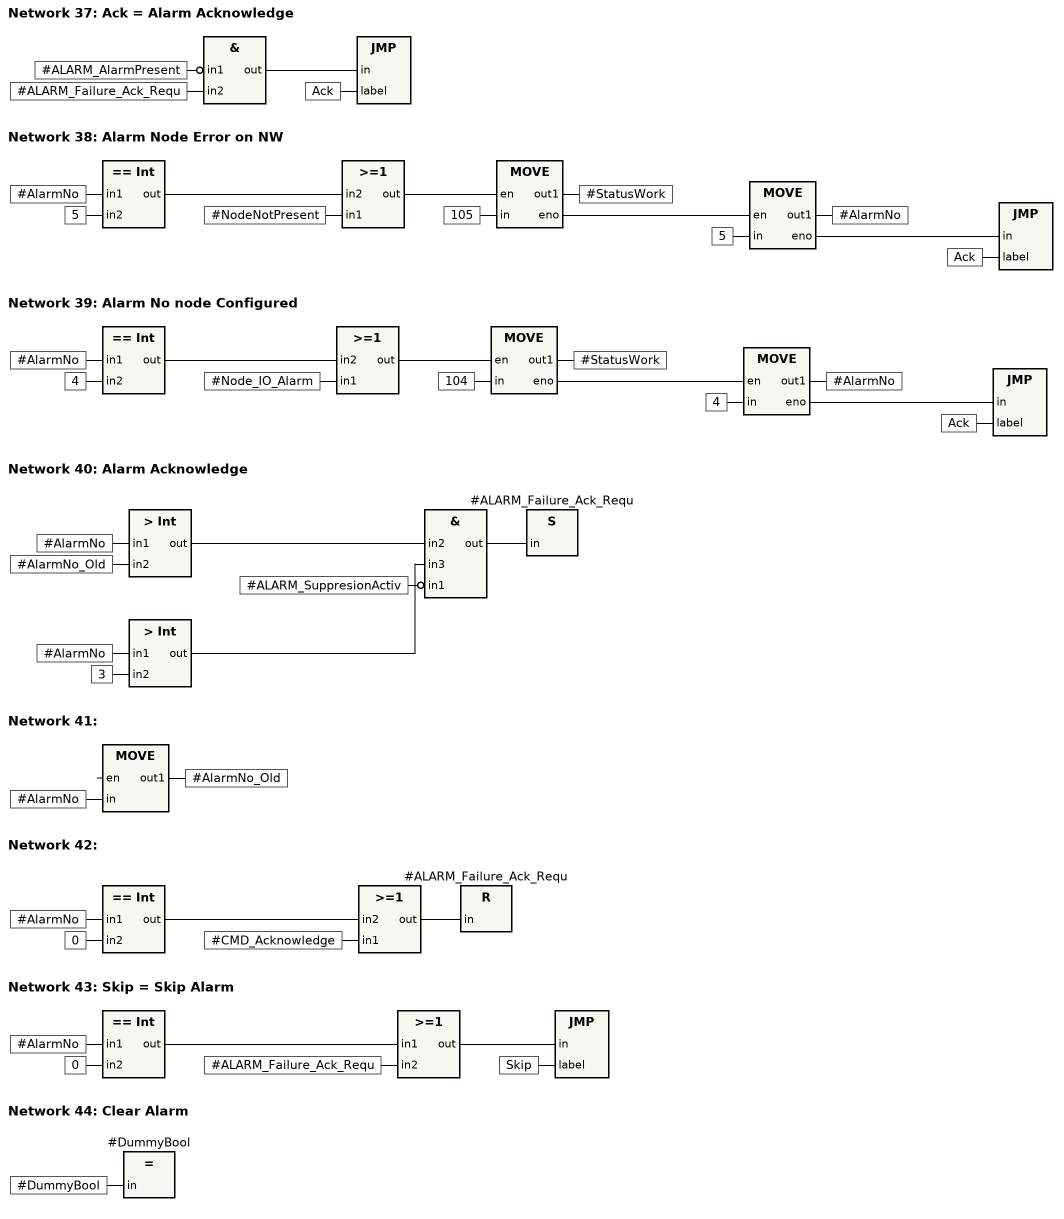
   IF NOT #ALARM_AlarmPresent AND #ALARM_Failure_Ack_Requ THEN GOTO Ack; END_IF;
END_REGION

REGION Network 38: Alarm Node Error on NW
   // ENO of a box is taken as its EN; it also drops when the box reports an error
   #_w1 := (#AlarmNo = 5) OR #NodeNotPresent;
   IF #_w1 THEN
       #StatusWork := 105;
       #AlarmNo := 5;
       GOTO Ack;
   END_IF;
END_REGION

REGION Network 39: Alarm No node Configured
   // ENO of a box is taken as its EN; it also drops when the box reports an error
   #_w1 := (#AlarmNo = 4) OR #Node_IO_Alarm;
   IF #_w1 THEN
       #StatusWork := 104;
       #AlarmNo := 4;
       GOTO Ack;
   END_IF;
END_REGION

REGION Network 40: Alarm Acknowledge
   Ack:
   IF (#AlarmNo > #AlarmNo_Old) AND (#AlarmNo > 3) AND NOT #ALARM_SuppresionActiv THEN
       #ALARM_Failure_Ack_Requ := TRUE;
   END_IF;
END_REGION

REGION Network 41
   #AlarmNo_Old := #AlarmNo;
END_REGION

REGION Network 42
   IF (#AlarmNo = 0) OR #CMD_Acknowledge THEN #ALARM_Failure_Ack_Requ := FALSE; END_IF;
END_REGION

REGION Network 43: Skip = Skip Alarm
   IF (#AlarmNo = 0) OR #ALARM_Failure_Ack_Requ THEN GOTO Skip; END_IF;
END_REGION

REGION Network 44: Clear Alarm
   Clr:
   #DummyBool := #DummyBool;
END_REGION

REGION Network 45
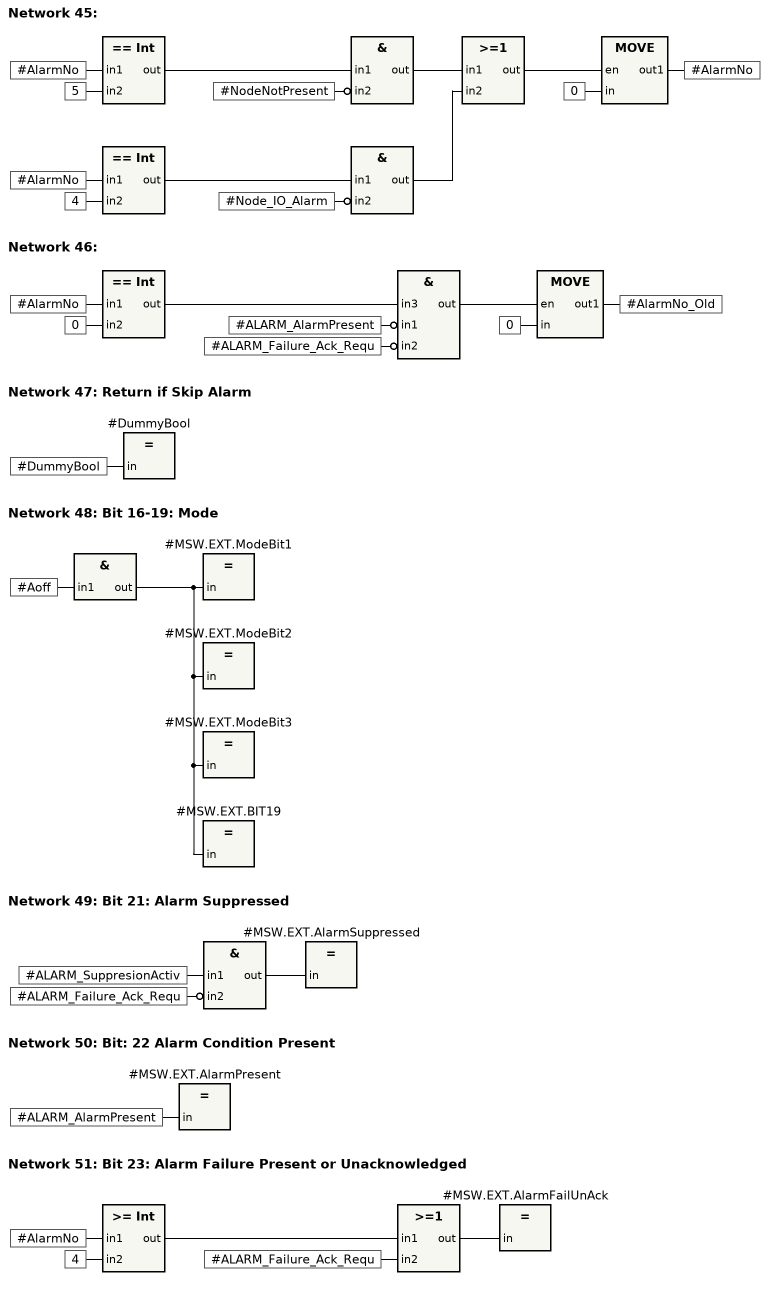
   IF ((#AlarmNo = 5) AND NOT #NodeNotPresent) OR ((#AlarmNo = 4) AND NOT #Node_IO_Alarm) THEN
       #AlarmNo := 0;
   END_IF;
END_REGION

REGION Network 46
   IF (#AlarmNo = 0) AND NOT #ALARM_AlarmPresent AND NOT #ALARM_Failure_Ack_Requ THEN
       #AlarmNo_Old := 0;
   END_IF;
END_REGION

REGION Network 47: Return if Skip Alarm
   Skip:
   #DummyBool := #DummyBool;
END_REGION

REGION Network 48: Bit 16-19: Mode
   // 0 = Auto
   // 1= Single Start
   // 2 = Manual
   // 3= Local
   // 4= Test Mode
   #MSW.EXT.ModeBit1 := #Aoff;
   #MSW.EXT.ModeBit2 := #Aoff;
   #MSW.EXT.ModeBit3 := #Aoff;
   #MSW.EXT.BIT19 := #Aoff;
END_REGION

REGION Network 49: Bit 21: Alarm Suppressed
   #MSW.EXT.AlarmSuppressed := #ALARM_SuppresionActiv AND NOT #ALARM_Failure_Ack_Requ;
END_REGION

REGION Network 50: Bit: 22 Alarm Condition Present
   #MSW.EXT.AlarmPresent := #ALARM_AlarmPresent;
END_REGION

REGION Network 51: Bit 23: Alarm Failure Present or Unacknowledged
   #MSW.EXT.AlarmFailUnAck := (#AlarmNo >= 4) OR #ALARM_Failure_Ack_Requ;
END_REGION

REGION Network 52: Bit 24: Alarm Warning Present Or Unacknowledged
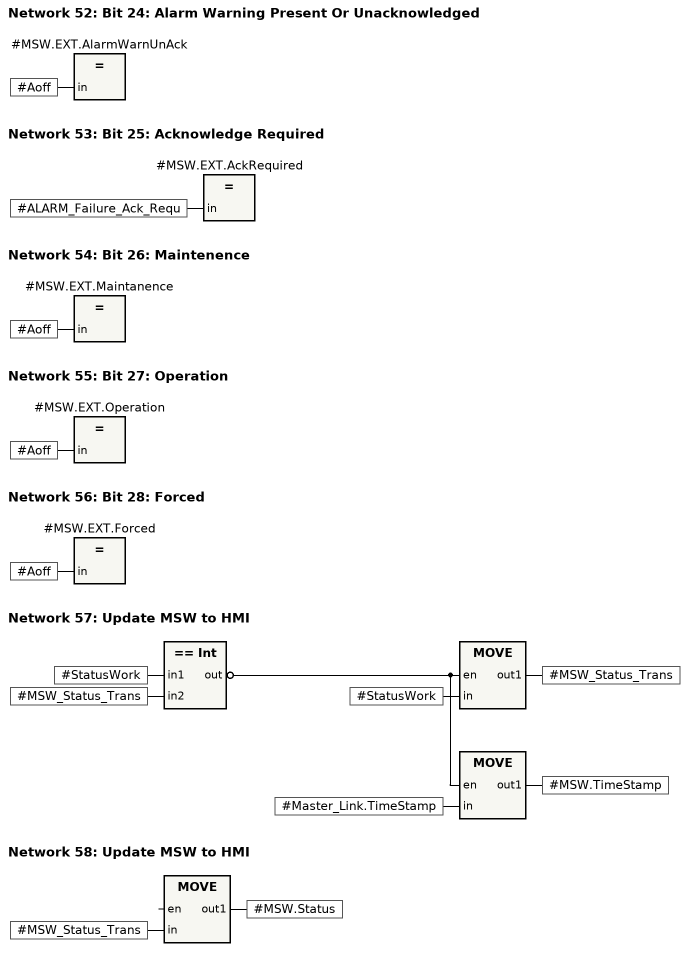
   #MSW.EXT.AlarmWarnUnAck := #Aoff;
END_REGION

REGION Network 53: Bit 25: Acknowledge Required
   #MSW.EXT.AckRequired := #ALARM_Failure_Ack_Requ;
END_REGION

REGION Network 54: Bit 26: Maintenence
   #MSW.EXT.Maintanence := #Aoff;
END_REGION

REGION Network 55: Bit 27: Operation
   #MSW.EXT.Operation := #Aoff;
END_REGION

REGION Network 56: Bit 28: Forced
   #MSW.EXT.Forced := #Aoff;
END_REGION

REGION Network 57: Update MSW to HMI
   #_w1 := NOT (#StatusWork = #MSW_Status_Trans);
   IF #_w1 THEN
       #MSW_Status_Trans := #StatusWork;
       #MSW.TimeStamp := #Master_Link.TimeStamp;
   END_IF;
END_REGION

REGION Network 58: Update MSW to HMI
   #MSW.Status := #MSW_Status_Trans;
END_REGION
END_FUNCTION_BLOCK

FUNCTION_BLOCK "ACESYS_SEND"   // FB225, FBD
TITLE = ACESYS V8.0 - Build 003 - SEND FUNCTION BLOCK
{ S7_Optimized_Access := 'TRUE' }
VERSION : 0.1
   VAR_INPUT
      Primary_EN : Bool;   // Enable Primary Link
      Primary_ID : Word;   // Valid from W#16#0001 to W#16#0FFF
      Primary_DEV_ID : Byte;   // 1 = Onboard (X1), 2 = Onboard (X2), 3 = Onboard (X3), 10 = External Cards
      Primary_ACT : Bool;   // ACTIVE=1; PASSIVE=0
      Primary_IP_ADDR1 : Int;   // Primary IP Address
      Primary_IP_ADDR2 : Int;   // Primary IP Address
      Primary_IP_ADDR3 : Int;   // Primary IP Address
      Primary_IP_ADDR4 : Int;   // Primary IP Address
      Primary_LOC_RS : Byte := BYTE#16#02;   // Primary Local Rack/Slot
      Primary_CP_RS : Byte;   // Primary CP Rack/Slot
      Primary_REM_RS : Byte := BYTE#16#02;   // Primary Remote Rack/Slot
      Secondary_EN : Bool;   // Enable Secondary Link
      Secondary_ID : Word;   // Valid from W#16#0001 to W#16#0FFF
      Secondary_DEV_ID : Byte;   // B#16#01-IM151-8PN, #02-CPU31x-2PN/DP, #03-CPU319-3PN/DP, #05-CPU41x-3PN/DP
      Secondary_ACT : Bool;
      Secondary_IP_ADDR1 : Int;   // Secondary IP Address
      Secondary_IP_ADDR2 : Int;   // Secondary IP Address
      Secondary_IP_ADDR3 : Int;   // Secondary IP Address
      Secondary_IP_ADDR4 : Int;   // Secondary IP Address
      Secondary_LOC_RS : Byte := BYTE#16#02;   // Secondary Local Rack/Slot
      Secondary_CP_RS : Byte;   // Secondary CP Rack/Slot
      Secondary_REM_RS : Byte := BYTE#16#02;   // Secondary Remote Rack/Slot
      DATA : "ACESYS_PlcToPLC";
      MASTER_LINK : "ACESYS_MASTER_LINK";
   END_VAR
   VAR_OUTPUT
      Primary_Comm_OK : Bool;   // Primary Communication OK
      Primary_Conn_St : Word;   // Primary Connection Status
      Primary_Send_St : Word;   // Primary Send Status
      Secondary_Comm_Ok : Bool;   // Secondary Communication OK
      Secondary_Conn_St : Word;   // Secondary Connection Status
      Secondary_Send_St : Word;   // Secondary Send Status
      MSW : "ACESYS_HMI_STAT_32T";
   END_VAR
   VAR
      BlockInfo : Struct
         Ace_Version : Int;   // Acesys Block Version Number
         Ace_BuildNo : Int;   // Acesys Block Build Number
         DB_Number : Int;   // Block Instance DB Number
      END_STRUCT;
      FP_CMD : Struct   // Faceplate Commands
         Spare_08 : Bool;
         Spare_09 : Bool;
         Spare_10 : Bool;
         Spare_11 : Bool;
         Spare_12 : Bool;
         Spare_13 : Bool;
         Spare_14 : Bool;
         AckAlarm : Bool;   // Alarm Acknowledge
         Spare_00 : Bool;
         Spare_01 : Bool;
         Spare_02 : Bool;
         Spare_03 : Bool;
         Spare_04 : Bool;
         Spare_05 : Bool;
         Spare_06 : Bool;
         Spare_07 : Bool;
      END_STRUCT;
      PRIM_T_SEND : TSEND;
      PRIM_T_CONN : TCON;
      PRIM_T_DISC : TDISCON;
      PRIM_T_PARAM : TCON_IP_RFC;
      PRIM_CONN_DATA : Struct
         REGISTERED : Bool;
         CONN_DONE : Bool;
         CONN_BUSY : Bool;
         CONN_ERROR : Bool;
         CONN_SETA : Bool;
         DISCONNECT : Bool;
         CONN_STATUS : Word;
         STATUS_SAV : Int;
         SEND_REQ : Bool;
         SEND_DONE : Bool;
         SEND_BUSY : Bool;
         SEND_ERROR : Bool;
         SEND_REQ_P : Bool;
         SEND_REQ_I : Bool;
         SEND_STATUS : Word;
         ABORT_REQ : Bool;
         ABORT_DONE : Bool;
         ABORT_BUSY : Bool;
         ABORT_ERROR : Bool;
         ABORT_REQ_I : Bool;
         ABORT_REQ_P : Bool;
         ABORT_STATUS : Word;
      END_STRUCT;
      SEC_T_SEND : TSEND;
      SEC_T_CONN : TCON;
      SEC_T_DISC : TDISCON;
      SEC_T_PARAM : TCON_IP_RFC;
      SEC_CONN_DATA : Struct
         REGISTERED : Bool;
         CONN_DONE : Bool;
         CONN_BUSY : Bool;
         CONN_ERROR : Bool;
         CONN_SETA : Bool;
         DISCONNECT : Bool;
         CONN_STATUS : Word;
         STATUS_SAV : Int;
         SEND_REQ : Bool;
         SEND_DONE : Bool;
         SEND_BUSY : Bool;
         SEND_ERROR : Bool;
         SEND_REQ_P : Bool;
         SEND_REQ_I : Bool;
         SEND_STATUS : Word;
         ABORT_REQ : Bool;
         ABORT_DONE : Bool;
         ABORT_BUSY : Bool;
         ABORT_ERROR : Bool;
         ABORT_REQ_I : Bool;
         ABORT_REQ_P : Bool;
         ABORT_STATUS : Word;
      END_STRUCT;
      TSAP16 : String[16];
      ID AT TSAP16 : Array[1..18] of Byte;
      Prim_String : String[16];
      Sec_String : String[16];
      Prim_INIT_COM : Bool;
      Sec_INIT_COM : Bool;
      Prim_En_ONS : Bool;
      Sec_En_ONS : Bool;
      Prim_Enabled_ONS : Bool;
      Sec_Enabled_ONS : Bool;
      SPECIFIED : Bool;
      Prim_ReCon_Active : Bool;   // Reconection Acive
      Sec_ReCon_Active : Bool;   // Reconection Acive
      Prim_SendReq_Dn : Bool;
      Sec_SendReq_Dn : Bool;
      Prim_EN : Bool;
      Sec_EN : Bool;
      Spare01 : Bool;
      Spare02 : Bool;
      Spare03 : Bool;
      Primary_ID_Old : Word;
      Secondary_ID_Old : Word;
      Prim_Con_TMR : TON_TIME;
      Prim_Del_ReCon : TON_TIME;   // Delay Before Auto ReConect
      Sec_Con_TMR : TON_TIME;
      Sec_Del_ReCon : TON_TIME;   // Delay Before Auto ReConect
      Prim_Com_OK : TON_TIME;
      Sec_Com_OK : TON_TIME;
      Prim_SendDelay : TON_TIME;
      Sec_SendDelay : TON_TIME;
      PRIM_EXT_HWID : GEOADDR;
      SEC_EXT_HWID : GEOADDR;
   END_VAR
   VAR_TEMP
      Aon : Bool;
      LOC_LEN : Int;
      REM_LEN : Int;
      TMP_INT : Int;
      LOC_RS : Int;
      TMP_RS : Int;
      TMP_DEV : Int;
      DummyBool : Bool;
      DummyDWord : DWord;
      DummyDInt : DInt;
      RET : Int;
      UDT_Length : Int;
      t_Zero : Int;
      b_Zero : Array[0..1] of Byte;
      SEND_DATA_Tmp : "ACESYS_PlcToPLC";
   END_VAR
   VAR_TEMP   // added for the SCL form of the ladder/FBD networks
      _w1 : Bool;
      _w2 : Bool;
      _w3 : Bool;
   END_VAR
BEGIN

REGION Network 1: Acesys Send Function Block based on Open Communication standard
   // Acesys Send Function Block based on Open Communication standard blocks FB63 and 
   // FB65 for ISO-on-TCP
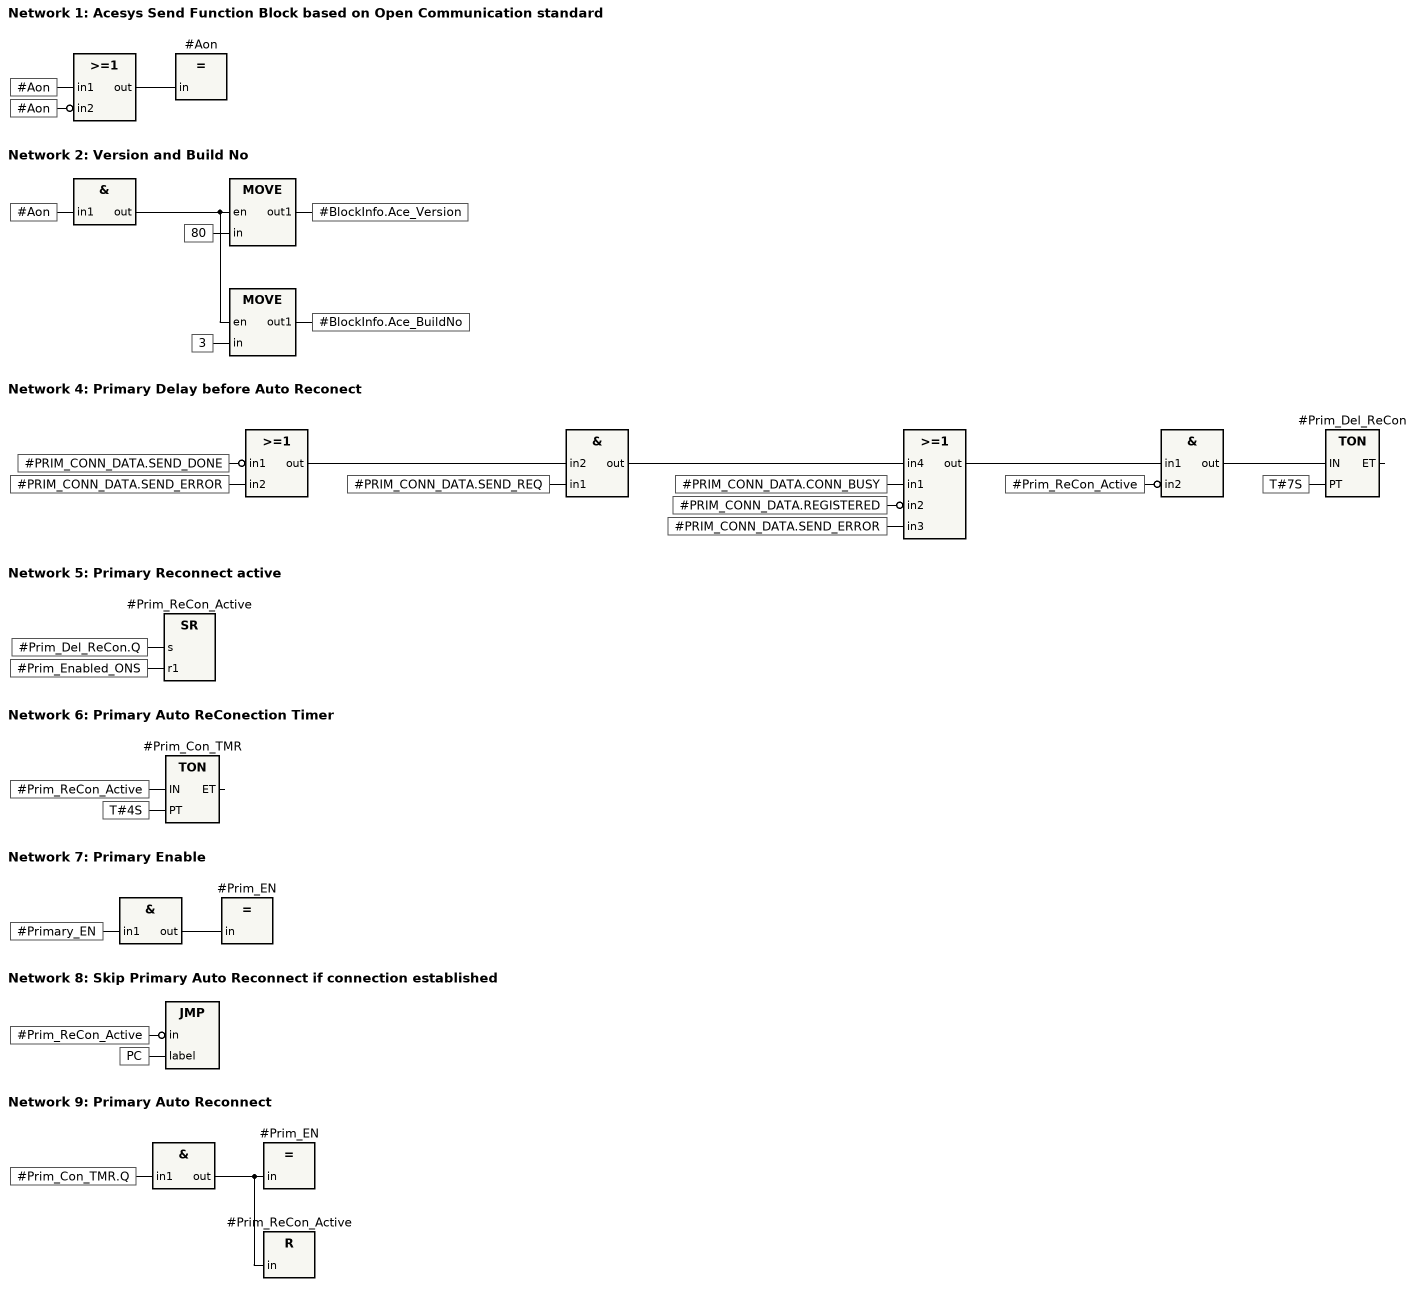
   #Aon := #Aon OR NOT #Aon;
END_REGION

REGION Network 2: Version and Build No
   IF #Aon THEN
       #BlockInfo.Ace_Version := 80;
       #BlockInfo.Ace_BuildNo := 3;
   END_IF;
END_REGION

REGION Network 3 (STL): Instance DB Number to Faceplate
         L     DINO;
         T     #BlockInfo.DB_Number;
END_REGION

REGION Network 4: Primary Delay before Auto Reconect
   #Prim_Del_ReCon(IN := (((NOT #PRIM_CONN_DATA.SEND_DONE OR #PRIM_CONN_DATA.SEND_ERROR) AND #PRIM_CONN_DATA.SEND_REQ) OR #PRIM_CONN_DATA.CONN_BUSY OR NOT #PRIM_CONN_DATA.REGISTERED OR #PRIM_CONN_DATA.SEND_ERROR) AND NOT #Prim_ReCon_Active,   // TON
                   PT := T#7S);
END_REGION

REGION Network 5: Primary Reconnect active
   IF #Prim_Del_ReCon.Q THEN
       #Prim_ReCon_Active := TRUE;   // SR flip-flop
   END_IF;
   IF #Prim_Enabled_ONS THEN #Prim_ReCon_Active := FALSE; END_IF;
END_REGION

REGION Network 6: Primary Auto ReConection Timer
   #Prim_Con_TMR(IN := #Prim_ReCon_Active, PT := T#4S);   // TON
END_REGION

REGION Network 7: Primary Enable
   #Prim_EN := #Primary_EN;
END_REGION

REGION Network 8: Skip Primary Auto Reconnect if connection established
   IF NOT #Prim_ReCon_Active THEN GOTO PC; END_IF;
END_REGION

REGION Network 9: Primary Auto Reconnect
   #Prim_EN := #Prim_Con_TMR.Q;
   IF #Prim_Con_TMR.Q THEN #Prim_ReCon_Active := FALSE; END_IF;
END_REGION

REGION Network 10: Set initial connection bit - Primary Link
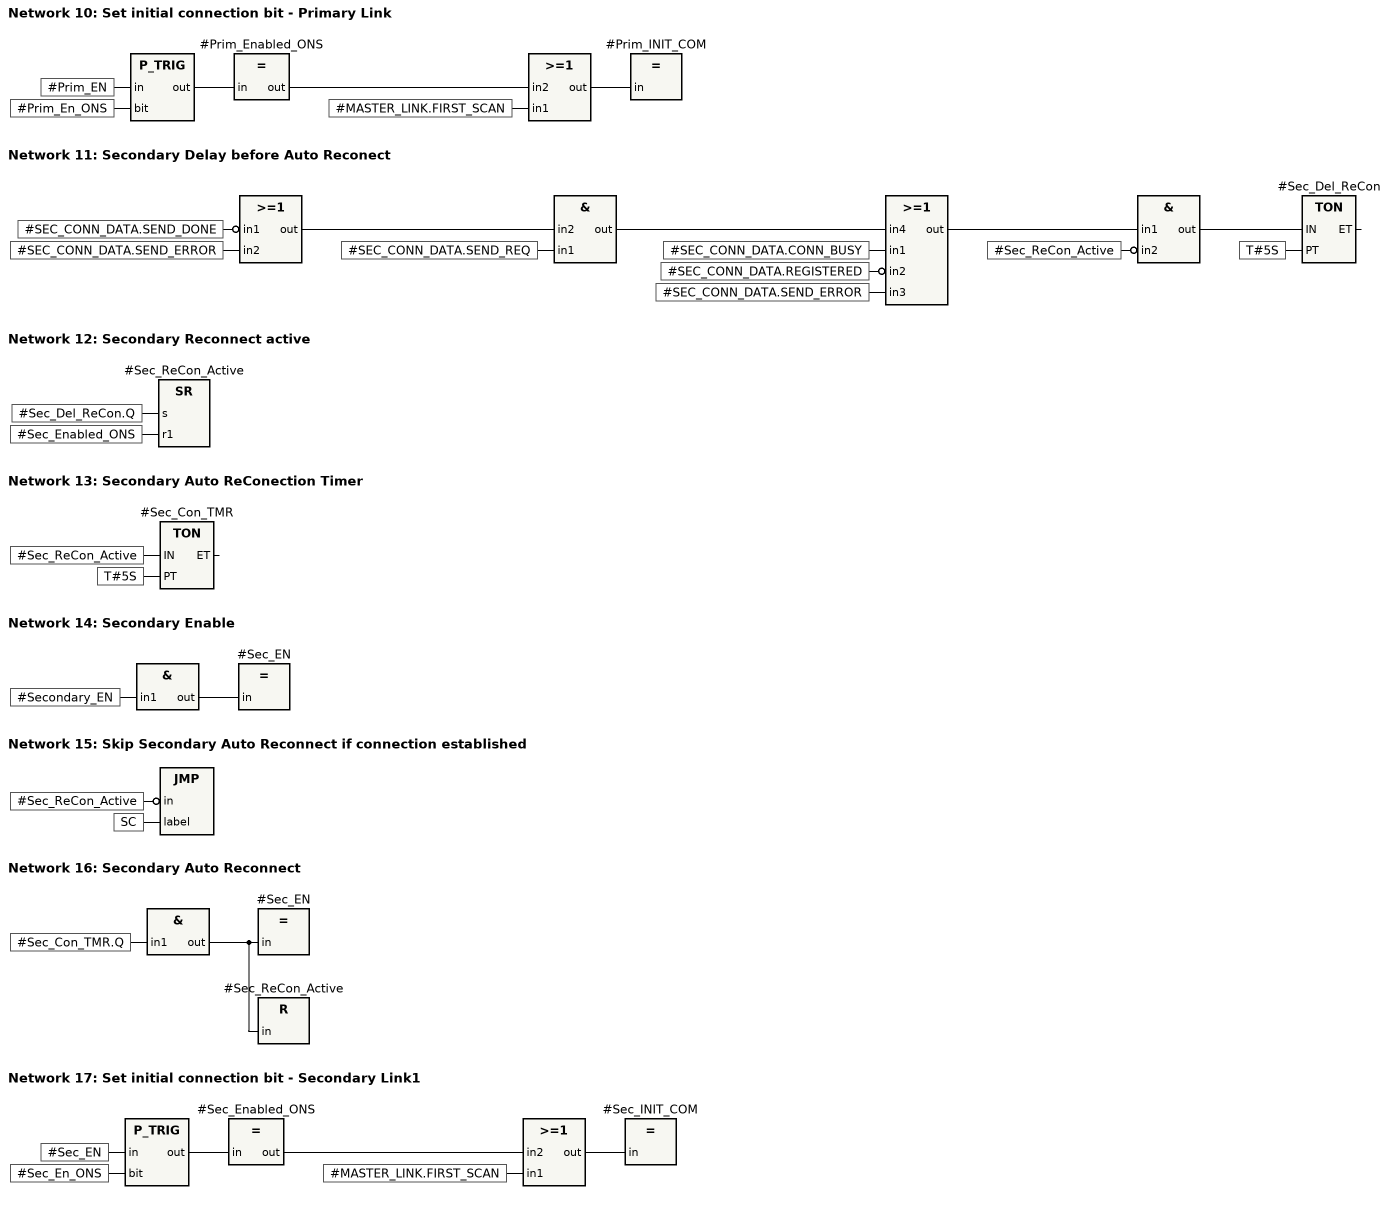
   PC:
   #_w1 := #Prim_EN AND NOT #Prim_En_ONS;   // rising edge
   #Prim_En_ONS := #Prim_EN;
   #Prim_Enabled_ONS := #_w1;
   #Prim_INIT_COM := #_w1 OR #MASTER_LINK.FIRST_SCAN;
END_REGION

REGION Network 11: Secondary Delay before Auto Reconect
   #Sec_Del_ReCon(IN := (((NOT #SEC_CONN_DATA.SEND_DONE OR #SEC_CONN_DATA.SEND_ERROR) AND #SEC_CONN_DATA.SEND_REQ) OR #SEC_CONN_DATA.CONN_BUSY OR NOT #SEC_CONN_DATA.REGISTERED OR #SEC_CONN_DATA.SEND_ERROR) AND NOT #Sec_ReCon_Active,   // TON
                  PT := T#5S);
END_REGION

REGION Network 12: Secondary Reconnect active
   IF #Sec_Del_ReCon.Q THEN
       #Sec_ReCon_Active := TRUE;   // SR flip-flop
   END_IF;
   IF #Sec_Enabled_ONS THEN #Sec_ReCon_Active := FALSE; END_IF;
END_REGION

REGION Network 13: Secondary Auto ReConection Timer
   #Sec_Con_TMR(IN := #Sec_ReCon_Active, PT := T#5S);   // TON
END_REGION

REGION Network 14: Secondary Enable
   #Sec_EN := #Secondary_EN;
END_REGION

REGION Network 15: Skip Secondary Auto Reconnect if connection established
   IF NOT #Sec_ReCon_Active THEN GOTO SC; END_IF;
END_REGION

REGION Network 16: Secondary Auto Reconnect
   #Sec_EN := #Sec_Con_TMR.Q;
   IF #Sec_Con_TMR.Q THEN #Sec_ReCon_Active := FALSE; END_IF;
END_REGION

REGION Network 17: Set initial connection bit - Secondary Link1
   SC:
   #_w1 := #Sec_EN AND NOT #Sec_En_ONS;   // rising edge
   #Sec_En_ONS := #Sec_EN;
   #Sec_Enabled_ONS := #_w1;
   #Sec_INIT_COM := #_w1 OR #MASTER_LINK.FIRST_SCAN;
END_REGION

REGION Network 18: Clear Bits to start initial connection and communication
   // Build002 - 27 March 2019 : Reset Condition PrimSendReq_Dn flag added
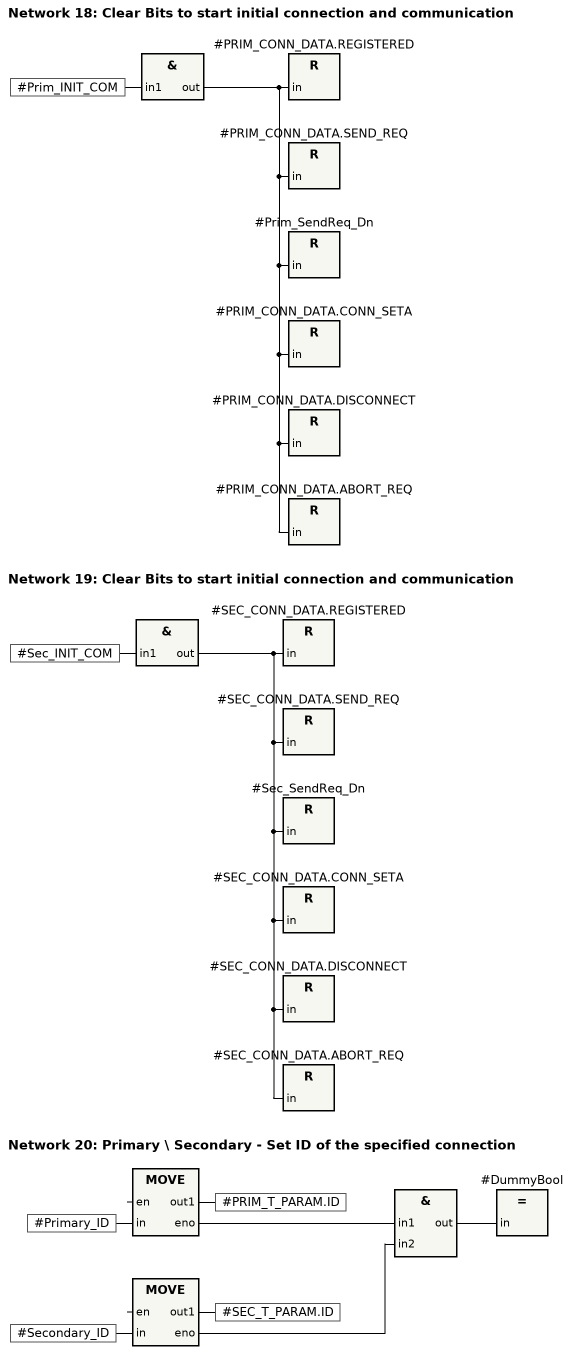
   IF #Prim_INIT_COM THEN
       #PRIM_CONN_DATA.REGISTERED := FALSE;
       #PRIM_CONN_DATA.SEND_REQ := FALSE;
       #Prim_SendReq_Dn := FALSE;
       #PRIM_CONN_DATA.CONN_SETA := FALSE;
       #PRIM_CONN_DATA.DISCONNECT := FALSE;
       #PRIM_CONN_DATA.ABORT_REQ := FALSE;
   END_IF;
END_REGION

REGION Network 19: Clear Bits to start initial connection and communication
   // Build002 - 27 March 2019 : Reset Condition SecSendReq_Dn flag added
   IF #Sec_INIT_COM THEN
       #SEC_CONN_DATA.REGISTERED := FALSE;
       #SEC_CONN_DATA.SEND_REQ := FALSE;
       #Sec_SendReq_Dn := FALSE;
       #SEC_CONN_DATA.CONN_SETA := FALSE;
       #SEC_CONN_DATA.DISCONNECT := FALSE;
       #SEC_CONN_DATA.ABORT_REQ := FALSE;
   END_IF;
END_REGION

REGION Network 20: Primary \ Secondary - Set ID of the specified connection
   // ENO of a box is taken as its EN; it also drops when the box reports an error
   #PRIM_T_PARAM.ID := #Primary_ID;
   #SEC_T_PARAM.ID := #Secondary_ID;
   #DummyBool := TRUE;
END_REGION

REGION Network 21: Primary \ Secondary - mode = 0x12 for ISO-on-TCP
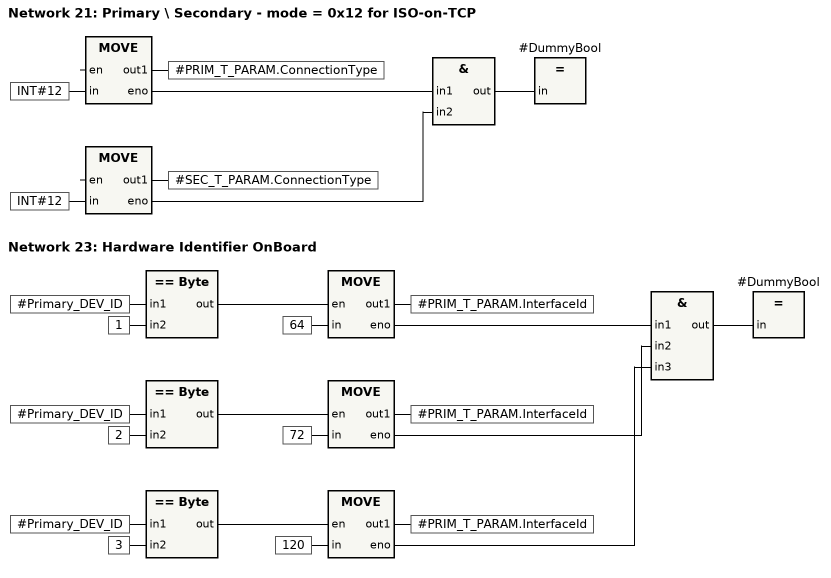
   // ENO of a box is taken as its EN; it also drops when the box reports an error
   #PRIM_T_PARAM.ConnectionType := INT#12;
   #SEC_T_PARAM.ConnectionType := INT#12;
   #DummyBool := TRUE;
END_REGION

REGION Network 22: <<<<<<<< PRIMARY >>>>>>>>
END_REGION

REGION Network 23: Hardware Identifier OnBoard
   // Build 003 viv-in 15 Feb 2022 -  X2 Port number corrected.
   #_w1 := #Primary_DEV_ID = 1;
   IF #_w1 THEN #PRIM_T_PARAM.InterfaceId := 64; END_IF;
   #_w2 := #Primary_DEV_ID = 2;
   IF #_w2 THEN #PRIM_T_PARAM.InterfaceId := 72; END_IF;
   #_w3 := #Primary_DEV_ID = 3;
   IF #_w3 THEN #PRIM_T_PARAM.InterfaceId := 120; END_IF;
   #DummyBool := #_w1 AND #_w2 AND #_w3;
END_REGION

REGION Network 24: Hardware Identifier External
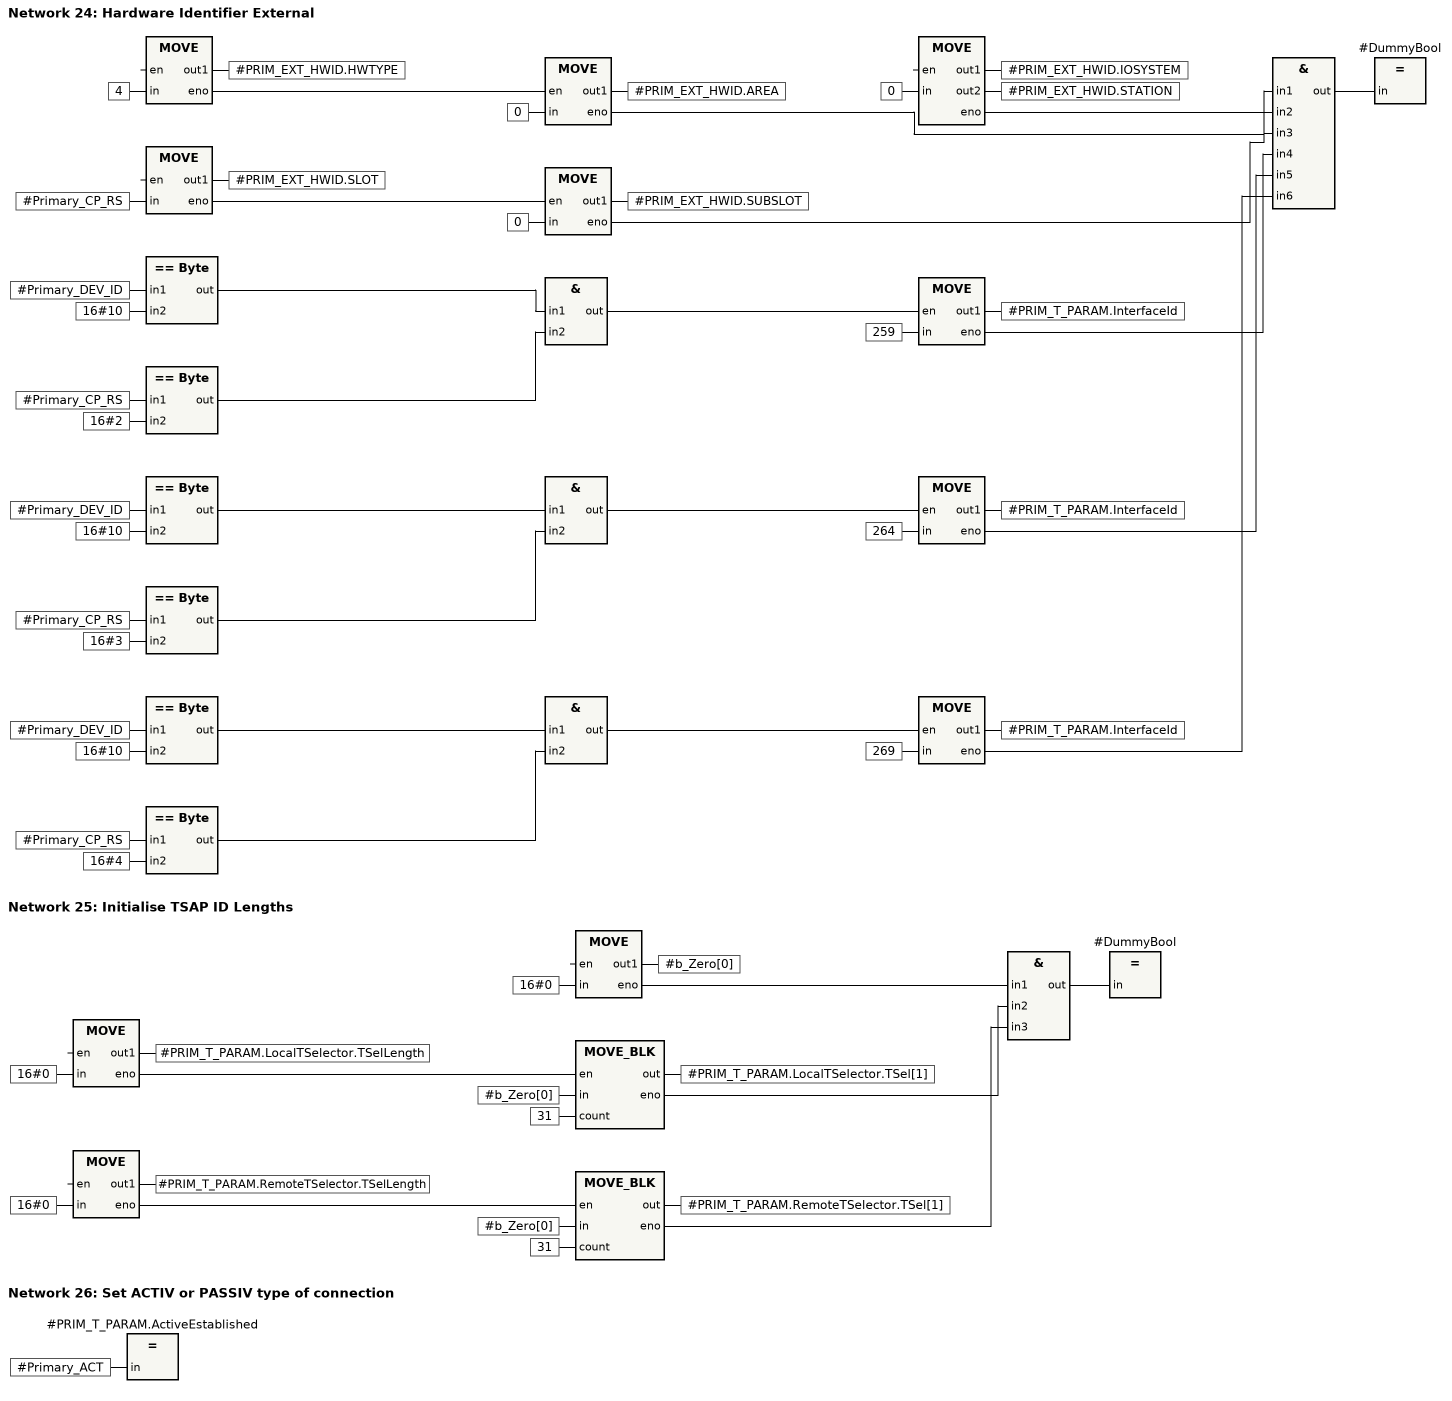
   #PRIM_EXT_HWID.HWTYPE := 4;
   #PRIM_EXT_HWID.AREA := 0;
   #PRIM_EXT_HWID.IOSYSTEM := 0;
   #PRIM_EXT_HWID.STATION := 0;
   #PRIM_EXT_HWID.SLOT := #Primary_CP_RS;
   #PRIM_EXT_HWID.SUBSLOT := 0;
   #_w1 := (#Primary_DEV_ID = 16#10) AND (#Primary_CP_RS = 16#2);
   IF #_w1 THEN #PRIM_T_PARAM.InterfaceId := 259; END_IF;
   #_w2 := (#Primary_DEV_ID = 16#10) AND (#Primary_CP_RS = 16#3);
   IF #_w2 THEN #PRIM_T_PARAM.InterfaceId := 264; END_IF;
   #_w3 := (#Primary_DEV_ID = 16#10) AND (#Primary_CP_RS = 16#4);
   IF #_w3 THEN #PRIM_T_PARAM.InterfaceId := 269; END_IF;
   #DummyBool := #_w1 AND #_w2 AND #_w3;
END_REGION

REGION Network 25: Initialise TSAP ID Lengths
   #b_Zero[0] := 16#0;
   #PRIM_T_PARAM.LocalTSelector.TSelLength := 16#0;
   MOVE_BLK(IN := #b_Zero[0], COUNT := 31, OUT => #PRIM_T_PARAM.LocalTSelector.TSel[1]);
   #PRIM_T_PARAM.RemoteTSelector.TSelLength := 16#0;
   MOVE_BLK(IN := #b_Zero[0], COUNT := 31, OUT => #PRIM_T_PARAM.RemoteTSelector.TSel[1]);
   #DummyBool := TRUE;
END_REGION

REGION Network 26: Set ACTIV or PASSIV type of connection
   // Receive Block Always Pasive
   #PRIM_T_PARAM.ActiveEstablished := #Primary_ACT;
END_REGION

REGION Network 27: Evaluate Rack/Slot being used for the leading bytes or none
   // 1) If R/S = 0 ---> no leading bytes are requested.
   // 2) If R/S # 0 ---> two leading bytes are required.
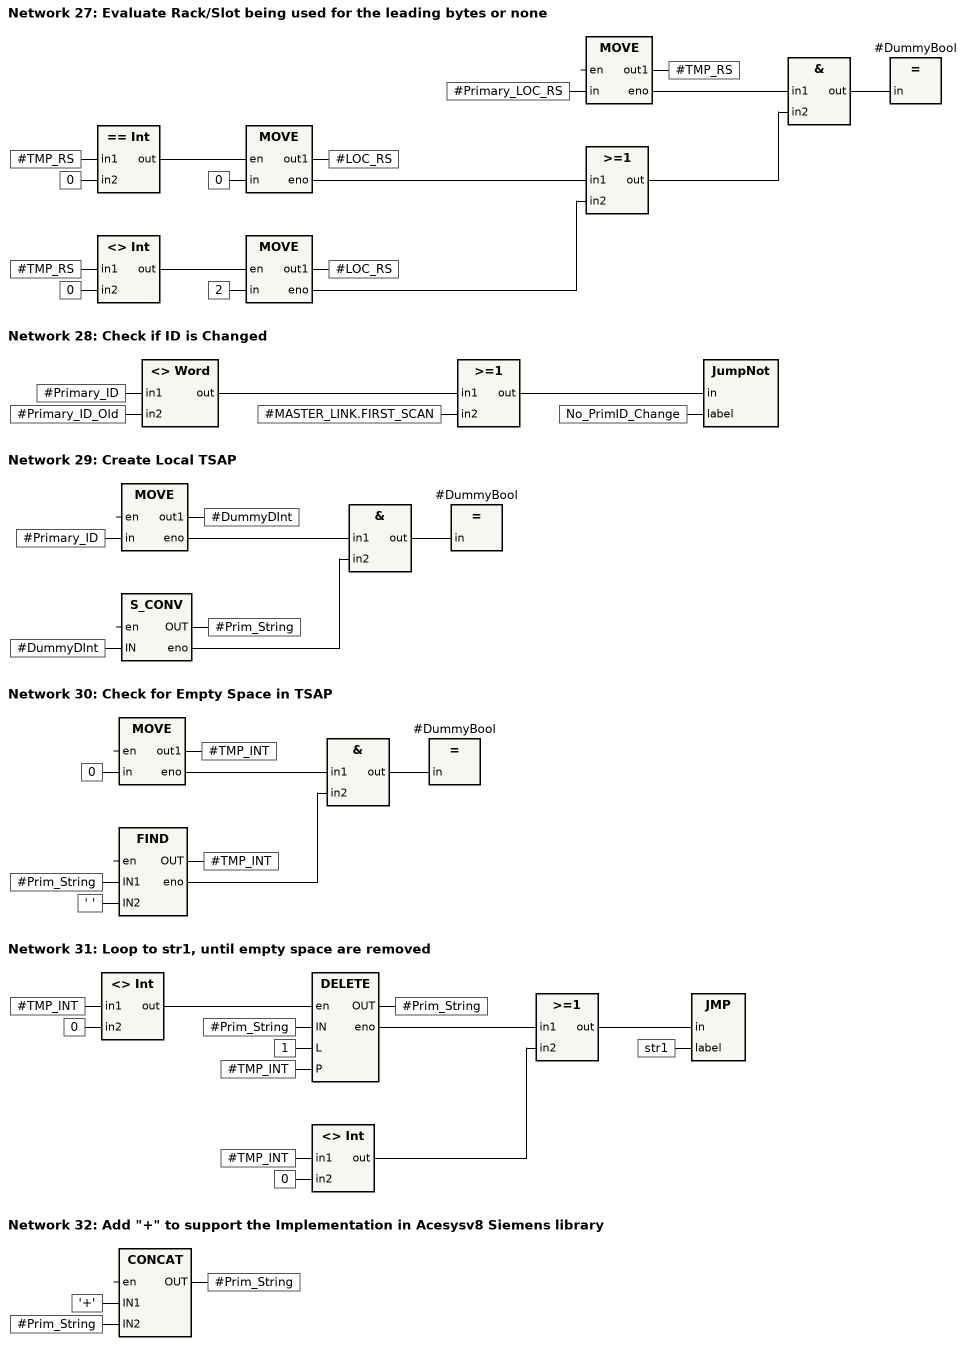
   // ENO of a box is taken as its EN; it also drops when the box reports an error
   #TMP_RS := #Primary_LOC_RS;
   #_w1 := #TMP_RS = 0;
   IF #_w1 THEN #LOC_RS := 0; END_IF;
   #_w2 := #TMP_RS <> 0;
   IF #_w2 THEN #LOC_RS := 2; END_IF;
   #DummyBool := #_w1 OR #_w2;
END_REGION

REGION Network 28: Check if ID is Changed
   // no SCL statement known for JumpNot: written as a call
   JumpNot(in := (#Primary_ID <> #Primary_ID_Old) OR #MASTER_LINK.FIRST_SCAN, label := No_PrimID_Change);
END_REGION

REGION Network 29: Create Local TSAP
   // Local TSAP = ID_Number
   // ENO of a box is taken as its EN; it also drops when the box reports an error
   #DummyDInt := #Primary_ID;
   #Prim_String := S_CONV(IN := #DummyDInt);
   #DummyBool := TRUE;
END_REGION

REGION Network 30: Check for Empty Space in TSAP
   str1:
   #TMP_INT := 0;
   #TMP_INT := FIND(IN1 := #Prim_String, IN2 := ' ');
   #DummyBool := TRUE;
END_REGION

REGION Network 31: Loop to str1, until empty space are removed
   #_w1 := #TMP_INT <> 0;
   IF #_w1 THEN #Prim_String := DELETE(IN := #Prim_String, L := 1, P := #TMP_INT); END_IF;
   IF #_w1 OR (#TMP_INT <> 0) THEN GOTO str1; END_IF;
END_REGION

REGION Network 32: Add "+" to support the Implementation in Acesysv8 Siemens library
   #Prim_String := CONCAT(IN1 := '+', IN2 := #Prim_String);
END_REGION

REGION Network 33: Set Primary_ID_Old Temp
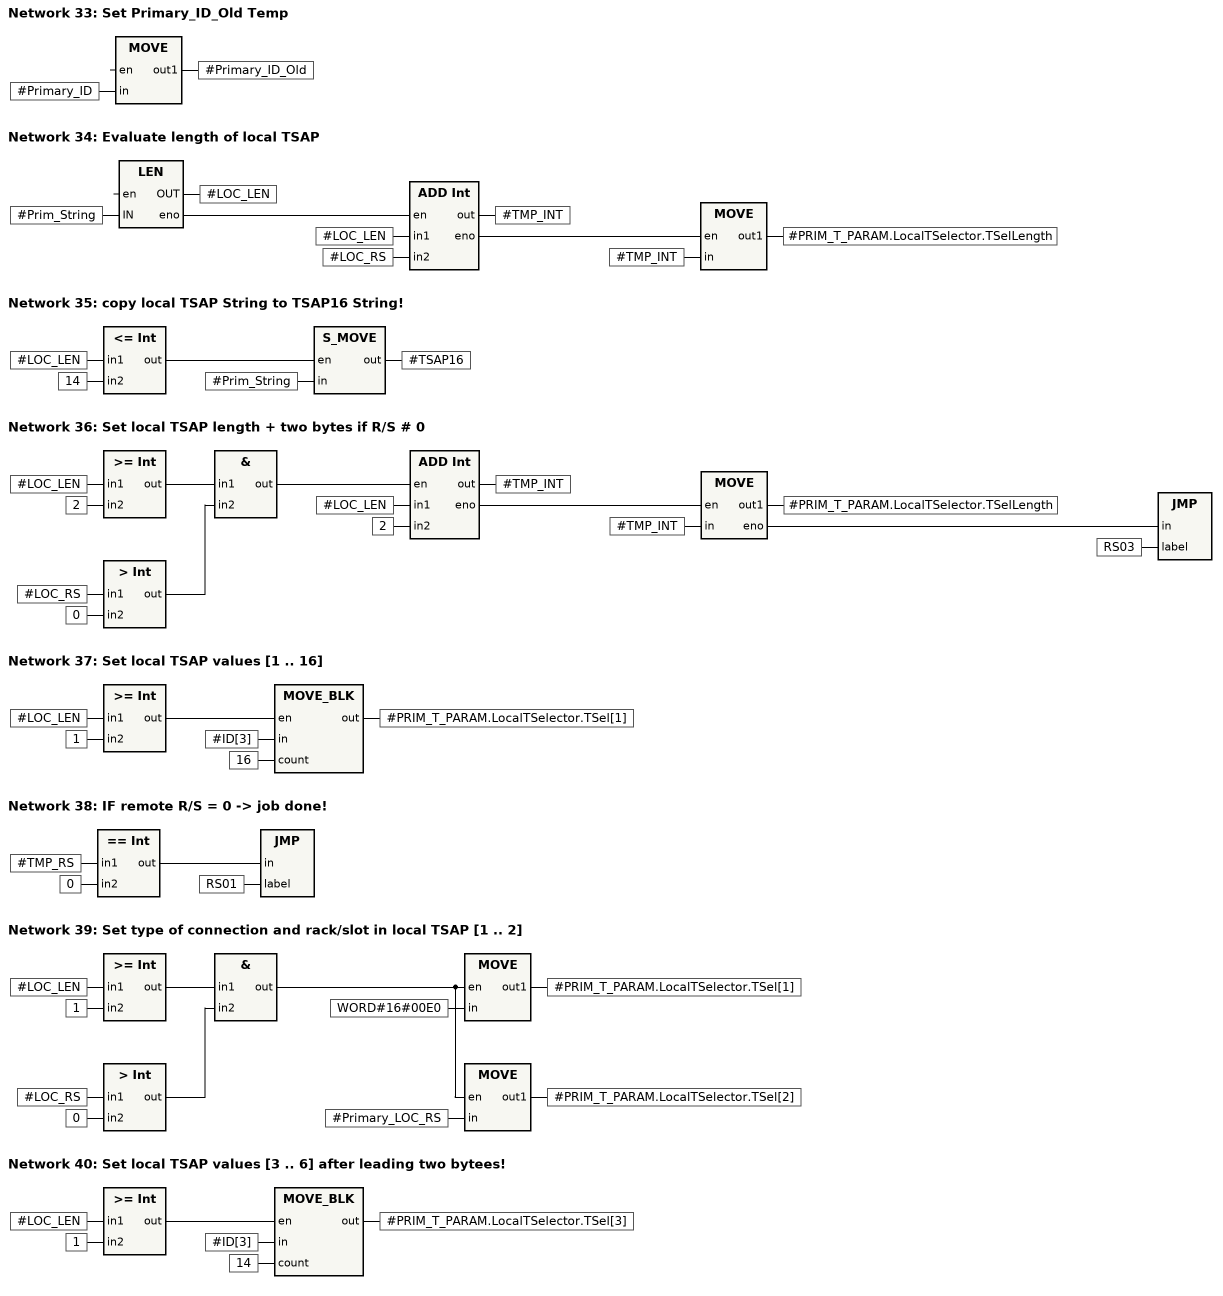
   No_PrimID_Change:
   #Primary_ID_Old := #Primary_ID;
END_REGION

REGION Network 34: Evaluate length of local TSAP
   // #TSAP.LOC_TSAP
   // ENO of a box is taken as its EN; it also drops when the box reports an error
   #LOC_LEN := LEN(IN := #Prim_String);
   #TMP_INT := #LOC_LEN + #LOC_RS;
   #PRIM_T_PARAM.LocalTSelector.TSelLength := #TMP_INT;
END_REGION

REGION Network 35: copy local TSAP String to TSAP16 String!
   // #TSAP.LOC_TSAP
   IF #LOC_LEN <= 14 THEN #TSAP16 := #Prim_String; END_IF;
END_REGION

REGION Network 36: Set local TSAP length + two bytes if R/S # 0
   // ENO of a box is taken as its EN; it also drops when the box reports an error
   #_w1 := (#LOC_LEN >= 2) AND (#LOC_RS > 0);
   IF #_w1 THEN
       #TMP_INT := #LOC_LEN + 2;
       #PRIM_T_PARAM.LocalTSelector.TSelLength := #TMP_INT;
       GOTO RS03;
   END_IF;
END_REGION

REGION Network 37: Set local TSAP values [1 .. 16]
   // Fill in the entire local TSAP (without leading bytes)
   IF #LOC_LEN >= 1 THEN
       MOVE_BLK(IN := #ID[3], COUNT := 16, OUT => #PRIM_T_PARAM.LocalTSelector.TSel[1]);
   END_IF;
END_REGION

REGION Network 38: IF remote R/S = 0 -> job done!
   IF #TMP_RS = 0 THEN GOTO RS01; END_IF;
END_REGION

REGION Network 39: Set type of connection and rack/slot in local TSAP [1 .. 2]
   // B#16#E0 -> type of connection 
   // B#16#02 -> rack/slot of CPU
   RS03:
   IF (#LOC_LEN >= 1) AND (#LOC_RS > 0) THEN
       #PRIM_T_PARAM.LocalTSelector.TSel[1] := WORD#16#00E0;
       #PRIM_T_PARAM.LocalTSelector.TSel[2] := #Primary_LOC_RS;
   END_IF;
END_REGION

REGION Network 40: Set local TSAP values [3 .. 6] after leading two bytees!
   IF #LOC_LEN >= 1 THEN
       MOVE_BLK(IN := #ID[3], COUNT := 14, OUT => #PRIM_T_PARAM.LocalTSelector.TSel[3]);
   END_IF;
END_REGION

REGION Network 41: REMOTE TSAP
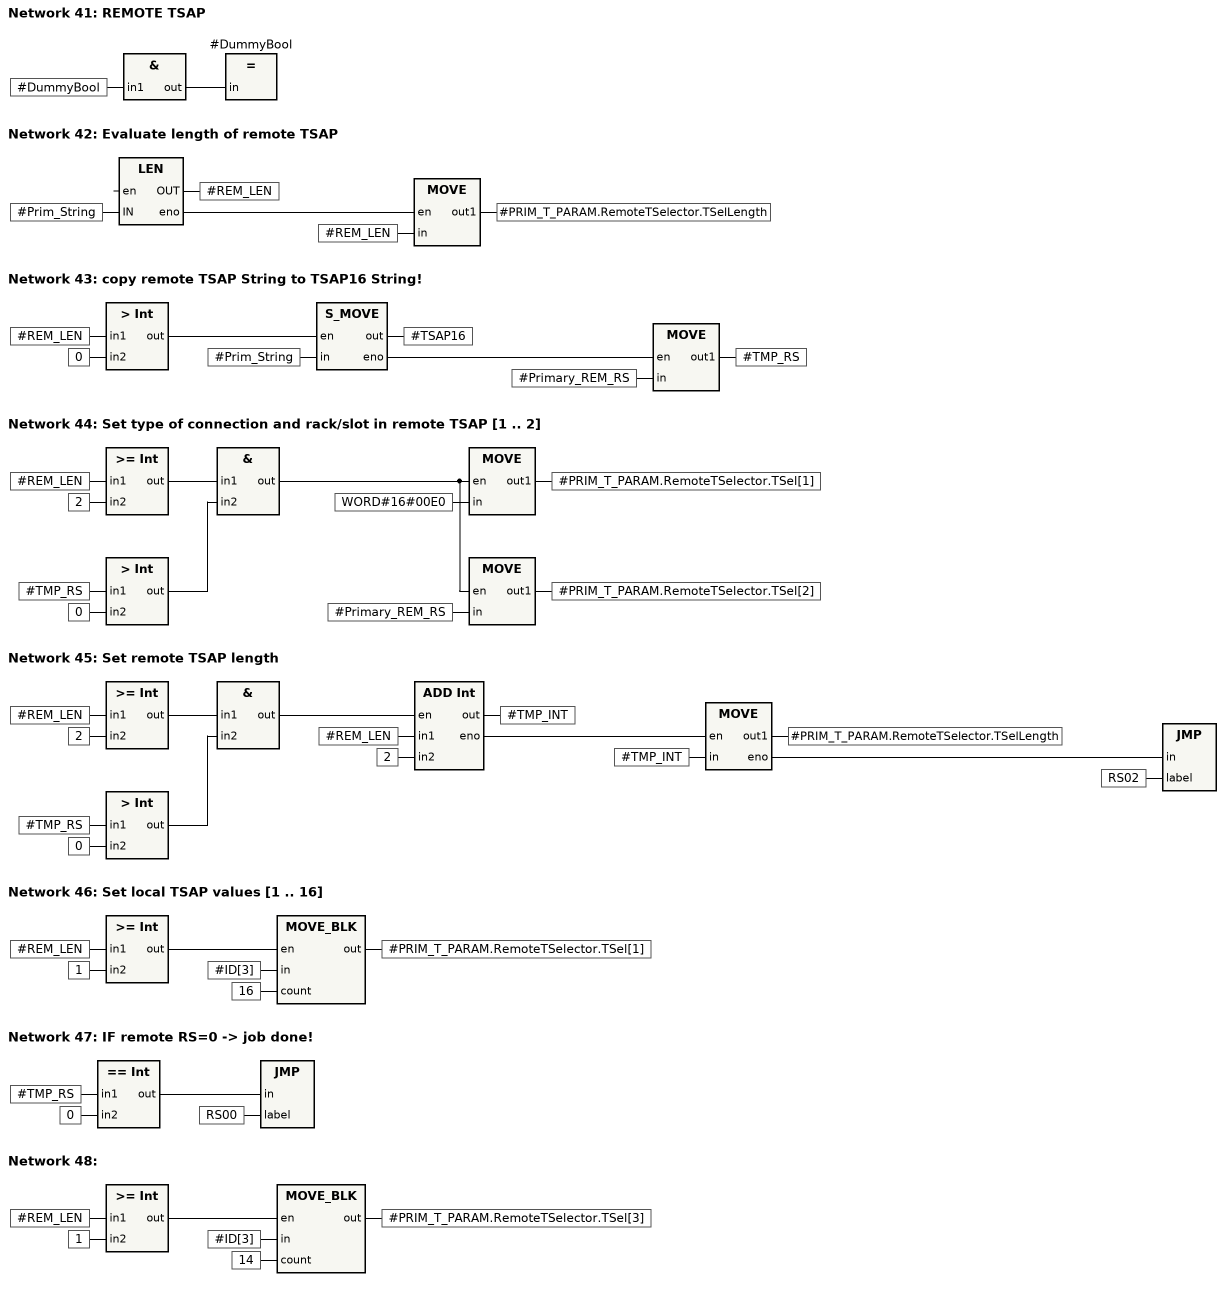
   RS01:
   #DummyBool := #DummyBool;
END_REGION

REGION Network 42: Evaluate length of remote TSAP
   // Remote TSAP = Local TSAP (DummyString1)
   #REM_LEN := LEN(IN := #Prim_String);
   #PRIM_T_PARAM.RemoteTSelector.TSelLength := #REM_LEN;
END_REGION

REGION Network 43: copy remote TSAP String to TSAP16 String!
   // Remote TSAP = Local TSAP (DummyString)
   IF #REM_LEN > 0 THEN
       #TSAP16 := #Prim_String;
       #TMP_RS := #Primary_REM_RS;
   END_IF;
END_REGION

REGION Network 44: Set type of connection and rack/slot in remote TSAP [1 .. 2]
   // B#16#E0 -> type of connection 
   // B#16#02 -> rack/slot of CPU
   IF (#REM_LEN >= 2) AND (#TMP_RS > 0) THEN
       #PRIM_T_PARAM.RemoteTSelector.TSel[1] := WORD#16#00E0;
       #PRIM_T_PARAM.RemoteTSelector.TSel[2] := #Primary_REM_RS;
   END_IF;
END_REGION

REGION Network 45: Set remote TSAP length
   // ENO of a box is taken as its EN; it also drops when the box reports an error
   #_w1 := (#REM_LEN >= 2) AND (#TMP_RS > 0);
   IF #_w1 THEN
       #TMP_INT := #REM_LEN + 2;
       #PRIM_T_PARAM.RemoteTSelector.TSelLength := #TMP_INT;
       GOTO RS02;
   END_IF;
END_REGION

REGION Network 46: Set local TSAP values [1 .. 16]
   // Fill in the entire local TSAP (without leading bytes)
   IF #REM_LEN >= 1 THEN
       MOVE_BLK(IN := #ID[3], COUNT := 16, OUT => #PRIM_T_PARAM.RemoteTSelector.TSel[1]);
   END_IF;
END_REGION

REGION Network 47: IF remote RS=0 -> job done!
   IF #TMP_RS = 0 THEN GOTO RS00; END_IF;
END_REGION

REGION Network 48
   RS02:
   IF #REM_LEN >= 1 THEN
       MOVE_BLK(IN := #ID[3], COUNT := 14, OUT => #PRIM_T_PARAM.RemoteTSelector.TSel[3]);
   END_IF;
END_REGION

REGION Network 49: Set length of the IP address if full-specified only !
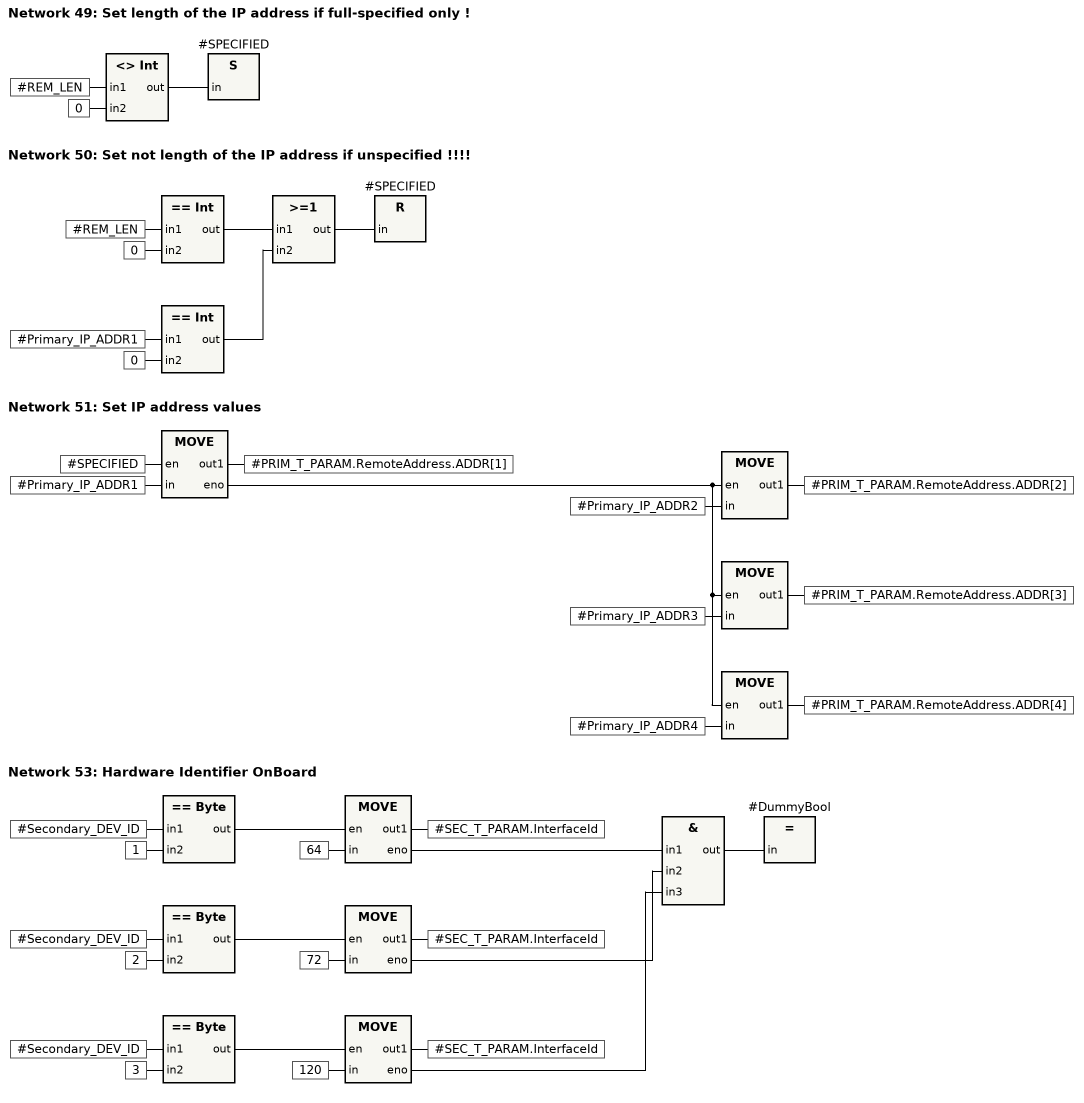
   RS00:
   IF #REM_LEN <> 0 THEN #SPECIFIED := TRUE; END_IF;
END_REGION

REGION Network 50: Set not length of the IP address if unspecified !!!!
   // The remote IP address must be zero if
   // 1) remote TSAP is unspecified, or
   // 2) IP address is set up with zero!
   IF (#REM_LEN = 0) OR (#Primary_IP_ADDR1 = 0) THEN #SPECIFIED := FALSE; END_IF;
END_REGION

REGION Network 51: Set IP address values
   // ENO of a box is taken as its EN; it also drops when the box reports an error
   IF #SPECIFIED THEN
       #PRIM_T_PARAM.RemoteAddress.ADDR[1] := #Primary_IP_ADDR1;
       #PRIM_T_PARAM.RemoteAddress.ADDR[2] := #Primary_IP_ADDR2;
       #PRIM_T_PARAM.RemoteAddress.ADDR[3] := #Primary_IP_ADDR3;
       #PRIM_T_PARAM.RemoteAddress.ADDR[4] := #Primary_IP_ADDR4;
   END_IF;
END_REGION

REGION Network 52: <<<<<<<<<<SECONDARY>>>>>>>>>>
END_REGION

REGION Network 53: Hardware Identifier OnBoard
   // Build 003 viv-in 15 Feb 2022 -  X2 Port number corrected.
   #_w1 := #Secondary_DEV_ID = 1;
   IF #_w1 THEN #SEC_T_PARAM.InterfaceId := 64; END_IF;
   #_w2 := #Secondary_DEV_ID = 2;
   IF #_w2 THEN #SEC_T_PARAM.InterfaceId := 72; END_IF;
   #_w3 := #Secondary_DEV_ID = 3;
   IF #_w3 THEN #SEC_T_PARAM.InterfaceId := 120; END_IF;
   #DummyBool := #_w1 AND #_w2 AND #_w3;
END_REGION

REGION Network 54: Hardware Identifier External
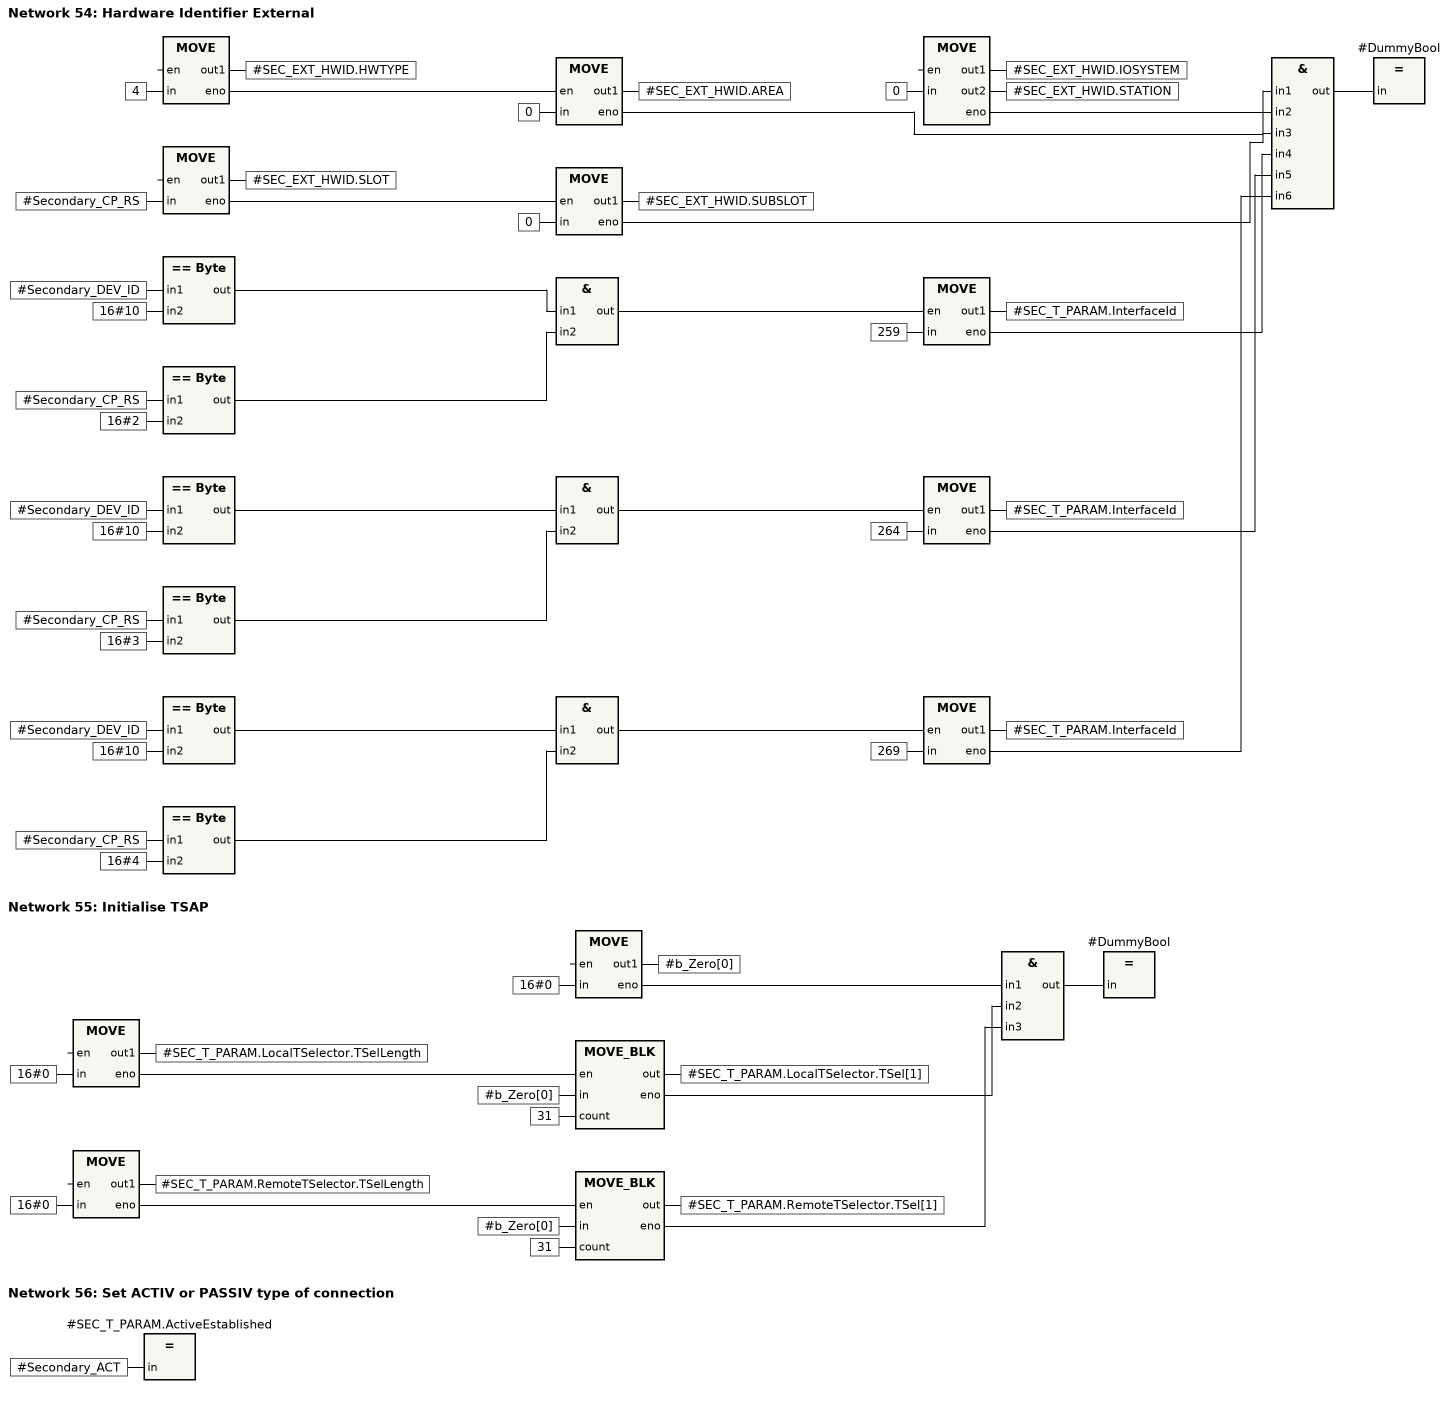
   #SEC_EXT_HWID.HWTYPE := 4;
   #SEC_EXT_HWID.AREA := 0;
   #SEC_EXT_HWID.IOSYSTEM := 0;
   #SEC_EXT_HWID.STATION := 0;
   #SEC_EXT_HWID.SLOT := #Secondary_CP_RS;
   #SEC_EXT_HWID.SUBSLOT := 0;
   #_w1 := (#Secondary_DEV_ID = 16#10) AND (#Secondary_CP_RS = 16#2);
   IF #_w1 THEN #SEC_T_PARAM.InterfaceId := 259; END_IF;
   #_w2 := (#Secondary_DEV_ID = 16#10) AND (#Secondary_CP_RS = 16#3);
   IF #_w2 THEN #SEC_T_PARAM.InterfaceId := 264; END_IF;
   #_w3 := (#Secondary_DEV_ID = 16#10) AND (#Secondary_CP_RS = 16#4);
   IF #_w3 THEN #SEC_T_PARAM.InterfaceId := 269; END_IF;
   #DummyBool := #_w1 AND #_w2 AND #_w3;
END_REGION

REGION Network 55: Initialise TSAP
   #b_Zero[0] := 16#0;
   #SEC_T_PARAM.LocalTSelector.TSelLength := 16#0;
   MOVE_BLK(IN := #b_Zero[0], COUNT := 31, OUT => #SEC_T_PARAM.LocalTSelector.TSel[1]);
   #SEC_T_PARAM.RemoteTSelector.TSelLength := 16#0;
   MOVE_BLK(IN := #b_Zero[0], COUNT := 31, OUT => #SEC_T_PARAM.RemoteTSelector.TSel[1]);
   #DummyBool := TRUE;
END_REGION

REGION Network 56: Set ACTIV or PASSIV type of connection
   // Send Block Always Active
   #SEC_T_PARAM.ActiveEstablished := #Secondary_ACT;
END_REGION

REGION Network 57: Evaluate Rack/Slot being used for the leading bytes or none
   // 1) If R/S = 0 ---> no leading bytes are requested.
   // 2) If R/S # 0 ---> two leading bytes are required.
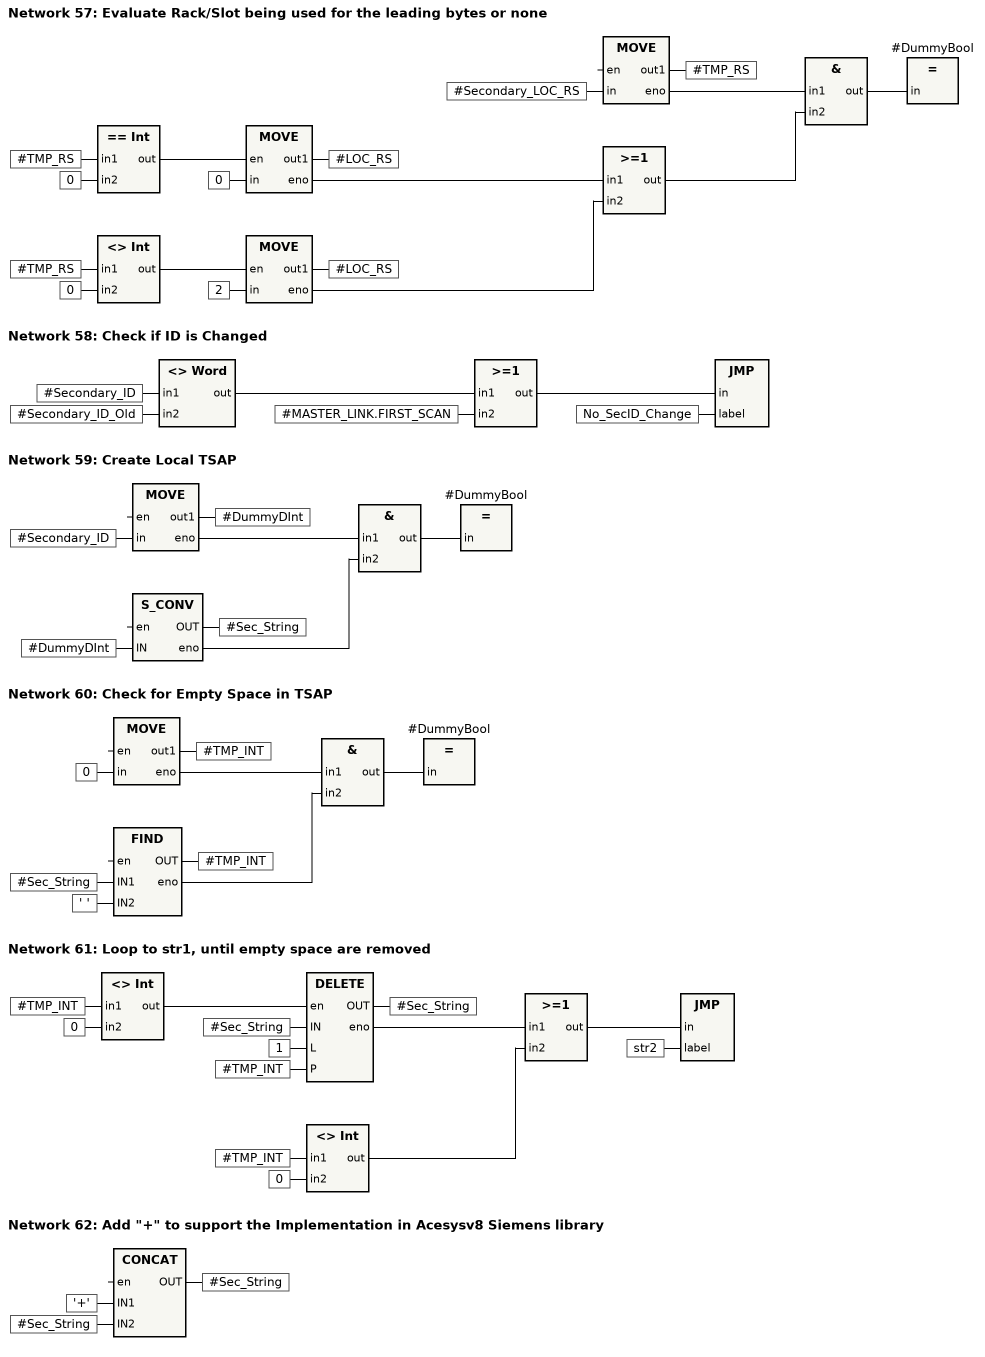
   // ENO of a box is taken as its EN; it also drops when the box reports an error
   #TMP_RS := #Secondary_LOC_RS;
   #_w1 := #TMP_RS = 0;
   IF #_w1 THEN #LOC_RS := 0; END_IF;
   #_w2 := #TMP_RS <> 0;
   IF #_w2 THEN #LOC_RS := 2; END_IF;
   #DummyBool := #_w1 OR #_w2;
END_REGION

REGION Network 58: Check if ID is Changed
   IF (#Secondary_ID <> #Secondary_ID_Old) OR #MASTER_LINK.FIRST_SCAN THEN GOTO No_SecID_Change; END_IF;
END_REGION

REGION Network 59: Create Local TSAP
   // Local TSAP = ID_Number
   // ENO of a box is taken as its EN; it also drops when the box reports an error
   #DummyDInt := #Secondary_ID;
   #Sec_String := S_CONV(IN := #DummyDInt);
   #DummyBool := TRUE;
END_REGION

REGION Network 60: Check for Empty Space in TSAP
   str2:
   #TMP_INT := 0;
   #TMP_INT := FIND(IN1 := #Sec_String, IN2 := ' ');
   #DummyBool := TRUE;
END_REGION

REGION Network 61: Loop to str1, until empty space are removed
   #_w1 := #TMP_INT <> 0;
   IF #_w1 THEN #Sec_String := DELETE(IN := #Sec_String, L := 1, P := #TMP_INT); END_IF;
   IF #_w1 OR (#TMP_INT <> 0) THEN GOTO str2; END_IF;
END_REGION

REGION Network 62: Add "+" to support the Implementation in Acesysv8 Siemens library
   #Sec_String := CONCAT(IN1 := '+', IN2 := #Sec_String);
END_REGION

REGION Network 63: Set Secondary_ID_Old Temp
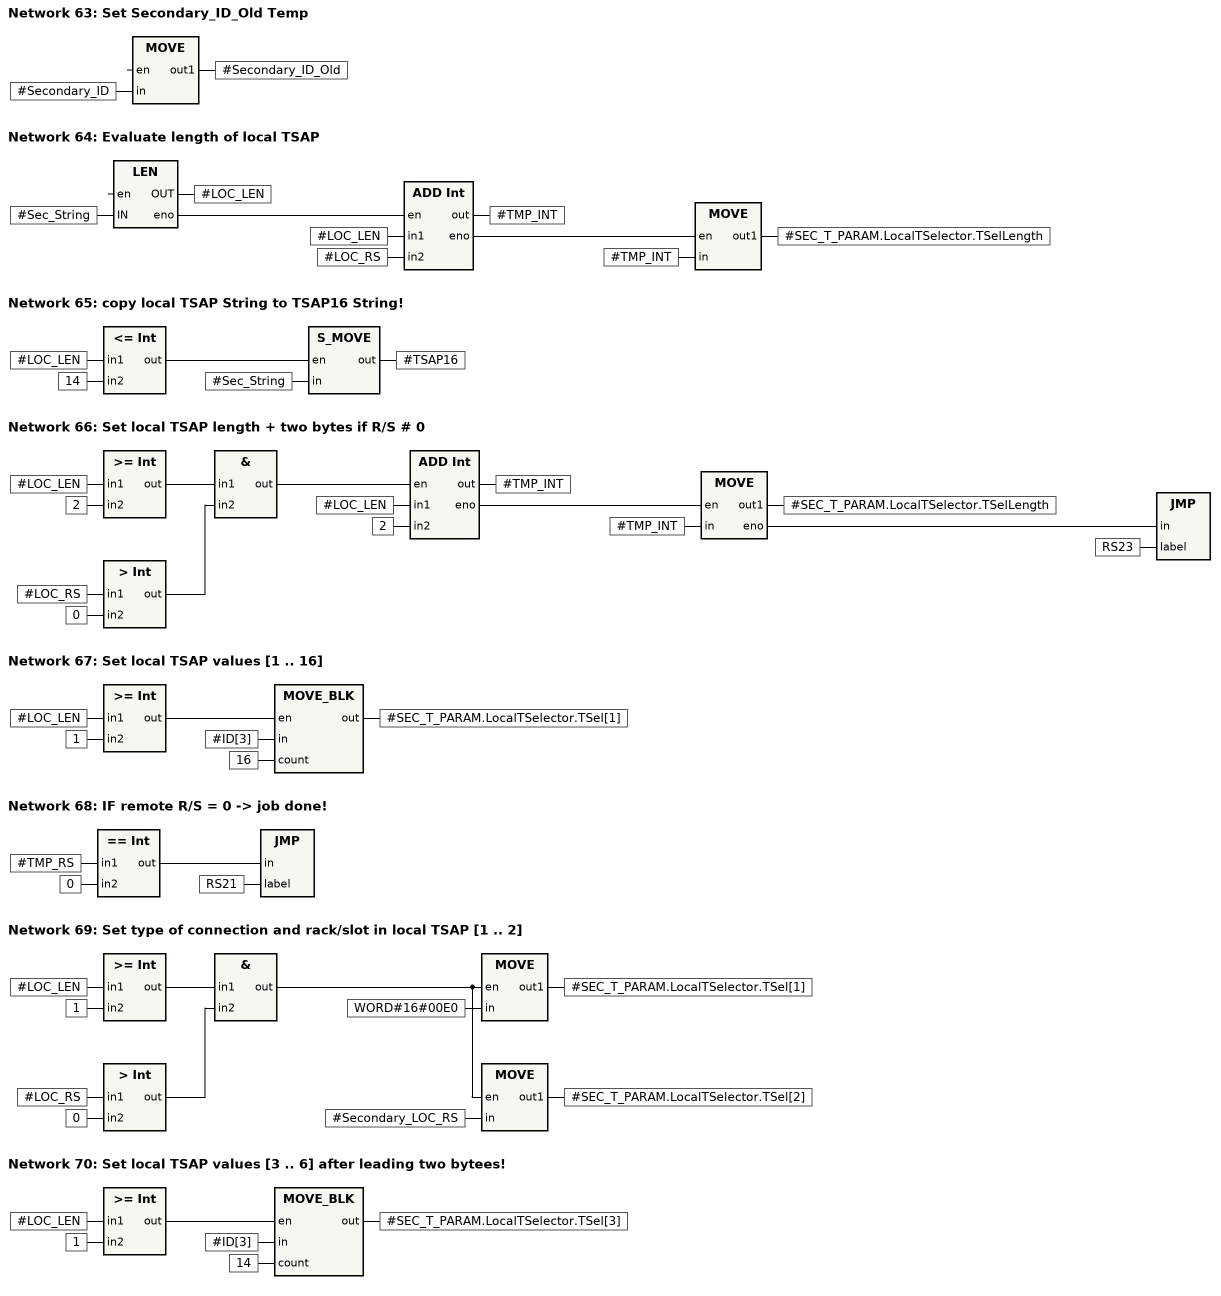
   No_SecID_Change:
   #Secondary_ID_Old := #Secondary_ID;
END_REGION

REGION Network 64: Evaluate length of local TSAP
   // #TSAP.LOC_TSAP
   // ENO of a box is taken as its EN; it also drops when the box reports an error
   #LOC_LEN := LEN(IN := #Sec_String);
   #TMP_INT := #LOC_LEN + #LOC_RS;
   #SEC_T_PARAM.LocalTSelector.TSelLength := #TMP_INT;
END_REGION

REGION Network 65: copy local TSAP String to TSAP16 String!
   // #TSAP.LOC_TSAP
   IF #LOC_LEN <= 14 THEN #TSAP16 := #Sec_String; END_IF;
END_REGION

REGION Network 66: Set local TSAP length + two bytes if R/S # 0
   // ENO of a box is taken as its EN; it also drops when the box reports an error
   #_w1 := (#LOC_LEN >= 2) AND (#LOC_RS > 0);
   IF #_w1 THEN
       #TMP_INT := #LOC_LEN + 2;
       #SEC_T_PARAM.LocalTSelector.TSelLength := #TMP_INT;
       GOTO RS23;
   END_IF;
END_REGION

REGION Network 67: Set local TSAP values [1 .. 16]
   // Fill in the entire local TSAP (without leading bytes)
   IF #LOC_LEN >= 1 THEN
       MOVE_BLK(IN := #ID[3], COUNT := 16, OUT => #SEC_T_PARAM.LocalTSelector.TSel[1]);
   END_IF;
END_REGION

REGION Network 68: IF remote R/S = 0 -> job done!
   IF #TMP_RS = 0 THEN GOTO RS21; END_IF;
END_REGION

REGION Network 69: Set type of connection and rack/slot in local TSAP [1 .. 2]
   // B#16#E0 -> type of connection 
   // B#16#02 -> rack/slot of CPU
   RS23:
   IF (#LOC_LEN >= 1) AND (#LOC_RS > 0) THEN
       #SEC_T_PARAM.LocalTSelector.TSel[1] := WORD#16#00E0;
       #SEC_T_PARAM.LocalTSelector.TSel[2] := #Secondary_LOC_RS;
   END_IF;
END_REGION

REGION Network 70: Set local TSAP values [3 .. 6] after leading two bytees!
   IF #LOC_LEN >= 1 THEN
       MOVE_BLK(IN := #ID[3], COUNT := 14, OUT => #SEC_T_PARAM.LocalTSelector.TSel[3]);
   END_IF;
END_REGION

REGION Network 71: <<<<<<< REMOTE TSAP >>>>>>>>
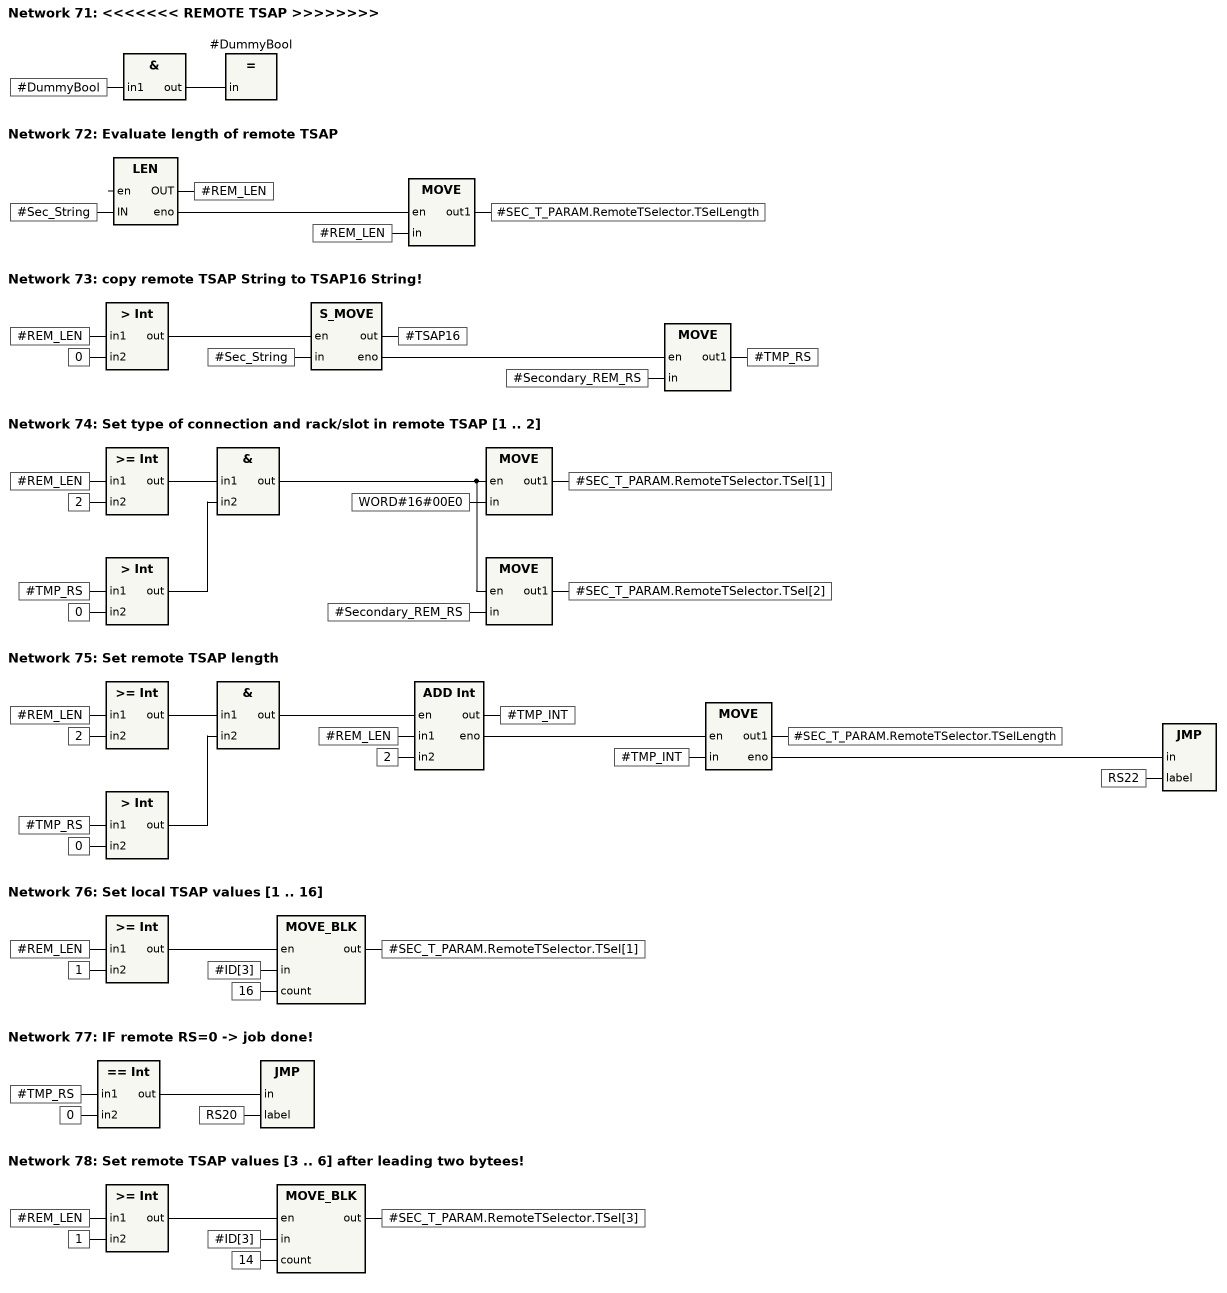
   RS21:
   #DummyBool := #DummyBool;
END_REGION

REGION Network 72: Evaluate length of remote TSAP
   // Remote TSAP = Local TSAP (DummyString1)
   #REM_LEN := LEN(IN := #Sec_String);
   #SEC_T_PARAM.RemoteTSelector.TSelLength := #REM_LEN;
END_REGION

REGION Network 73: copy remote TSAP String to TSAP16 String!
   // Remote TSAP = Local TSAP (DummyString)
   IF #REM_LEN > 0 THEN
       #TSAP16 := #Sec_String;
       #TMP_RS := #Secondary_REM_RS;
   END_IF;
END_REGION

REGION Network 74: Set type of connection and rack/slot in remote TSAP [1 .. 2]
   // B#16#E0 -> type of connection 
   // B#16#02 -> rack/slot of CPU
   IF (#REM_LEN >= 2) AND (#TMP_RS > 0) THEN
       #SEC_T_PARAM.RemoteTSelector.TSel[1] := WORD#16#00E0;
       #SEC_T_PARAM.RemoteTSelector.TSel[2] := #Secondary_REM_RS;
   END_IF;
END_REGION

REGION Network 75: Set remote TSAP length
   // ENO of a box is taken as its EN; it also drops when the box reports an error
   #_w1 := (#REM_LEN >= 2) AND (#TMP_RS > 0);
   IF #_w1 THEN
       #TMP_INT := #REM_LEN + 2;
       #SEC_T_PARAM.RemoteTSelector.TSelLength := #TMP_INT;
       GOTO RS22;
   END_IF;
END_REGION

REGION Network 76: Set local TSAP values [1 .. 16]
   // Fill in the entire local TSAP (without leading bytes)
   IF #REM_LEN >= 1 THEN
       MOVE_BLK(IN := #ID[3], COUNT := 16, OUT => #SEC_T_PARAM.RemoteTSelector.TSel[1]);
   END_IF;
END_REGION

REGION Network 77: IF remote RS=0 -> job done!
   IF #TMP_RS = 0 THEN GOTO RS20; END_IF;
END_REGION

REGION Network 78: Set remote TSAP values [3 .. 6] after leading two bytees!
   RS22:
   IF #REM_LEN >= 1 THEN
       MOVE_BLK(IN := #ID[3], COUNT := 14, OUT => #SEC_T_PARAM.RemoteTSelector.TSel[3]);
   END_IF;
END_REGION

REGION Network 79: Set length of the IP address if full-specified only !
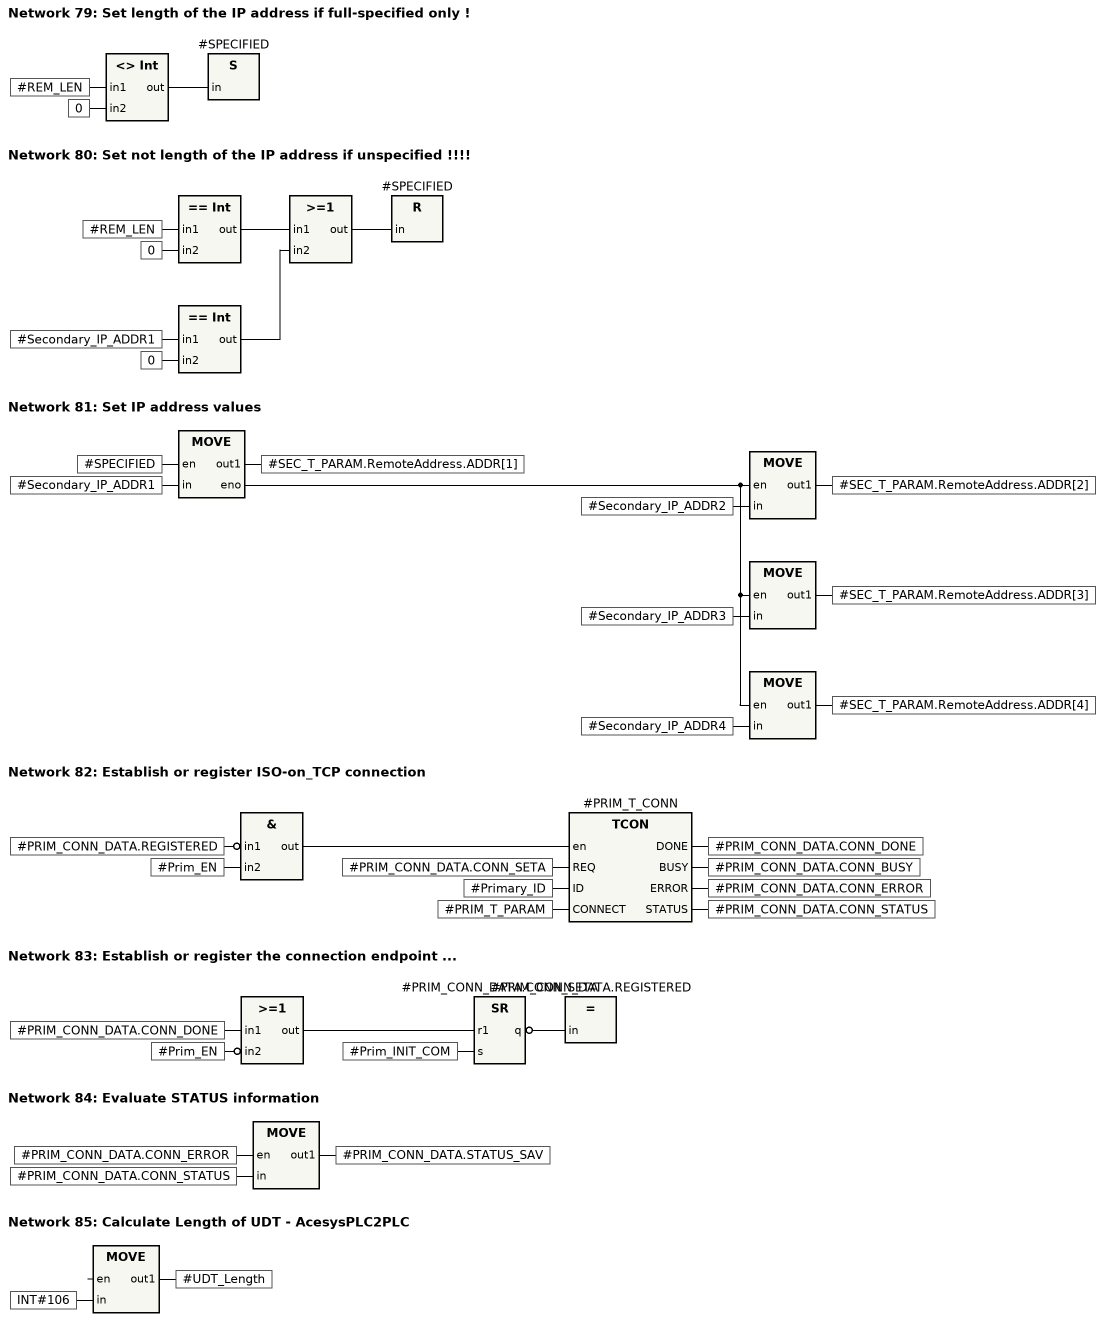
   RS20:
   IF #REM_LEN <> 0 THEN #SPECIFIED := TRUE; END_IF;
END_REGION

REGION Network 80: Set not length of the IP address if unspecified !!!!
   // The remote IP address must be zero if
   // 1) remote TSAP is unspecified, or
   // 2) IP address is set up with zero!
   IF (#REM_LEN = 0) OR (#Secondary_IP_ADDR1 = 0) THEN #SPECIFIED := FALSE; END_IF;
END_REGION

REGION Network 81: Set IP address values
   // ENO of a box is taken as its EN; it also drops when the box reports an error
   IF #SPECIFIED THEN
       #SEC_T_PARAM.RemoteAddress.ADDR[1] := #Secondary_IP_ADDR1;
       #SEC_T_PARAM.RemoteAddress.ADDR[2] := #Secondary_IP_ADDR2;
       #SEC_T_PARAM.RemoteAddress.ADDR[3] := #Secondary_IP_ADDR3;
       #SEC_T_PARAM.RemoteAddress.ADDR[4] := #Secondary_IP_ADDR4;
   END_IF;
END_REGION

REGION Network 82: Establish or register ISO-on_TCP connection
   // After the connection has been established, it is automatically monitored and 
   // maintained by the operating system of the CPU.
   // 
   // If the connection has been interrupted, by any line break or due to the remote 
   // communications partner, the active partner attempts to reestablish the 
   // connection.
   // 
   // Therefore, the FB 65 "TCON" may not be called again!
   IF NOT #PRIM_CONN_DATA.REGISTERED AND #Prim_EN THEN
       #PRIM_T_CONN(REQ := #PRIM_CONN_DATA.CONN_SETA,   // TCON
                    ID := #Primary_ID,
                    CONNECT := #PRIM_T_PARAM,
                    DONE => #PRIM_CONN_DATA.CONN_DONE,
                    BUSY => #PRIM_CONN_DATA.CONN_BUSY,
                    ERROR => #PRIM_CONN_DATA.CONN_ERROR,
                    STATUS => #PRIM_CONN_DATA.CONN_STATUS);
   END_IF;
END_REGION

REGION Network 83: Establish or register the connection endpoint ...
   // while startup phase (initial).
   // 
   // Indication of the connection status:
   // 
   // a) If the CPU may establish the specified connection after Stop/Run  
   // immediately, the variable "REGISTERED" indicates HIGH (=1).
   // 
   // b) If the CPU is not able to establish the specified connection after Stop/Run, 
   // the variable "REGISTERED" remains LOW(=0).
   // 
   // c) Note: If the instance DB is loaded by the user, the variable "REGISTERED" 
   // indicates HIGH, although the connection may not be established yet. 
   // However, the FB64 "TRCV" would indicate the STATUS=0x80C4, as long as the 
   // connection has not been established.
   IF #Prim_INIT_COM THEN
       #PRIM_CONN_DATA.CONN_SETA := TRUE;   // SR flip-flop
   END_IF;
   IF #PRIM_CONN_DATA.CONN_DONE OR NOT #Prim_EN THEN #PRIM_CONN_DATA.CONN_SETA := FALSE; END_IF;
   #PRIM_CONN_DATA.REGISTERED := NOT #PRIM_CONN_DATA.CONN_SETA;
END_REGION

REGION Network 84: Evaluate STATUS information
   // If ERROR occured then save STATUS!
   IF #PRIM_CONN_DATA.CONN_ERROR THEN #PRIM_CONN_DATA.STATUS_SAV := #PRIM_CONN_DATA.CONN_STATUS; END_IF;
END_REGION

REGION Network 85: Calculate Length of UDT - AcesysPLC2PLC
   #UDT_Length := INT#106;
END_REGION

REGION Network 86
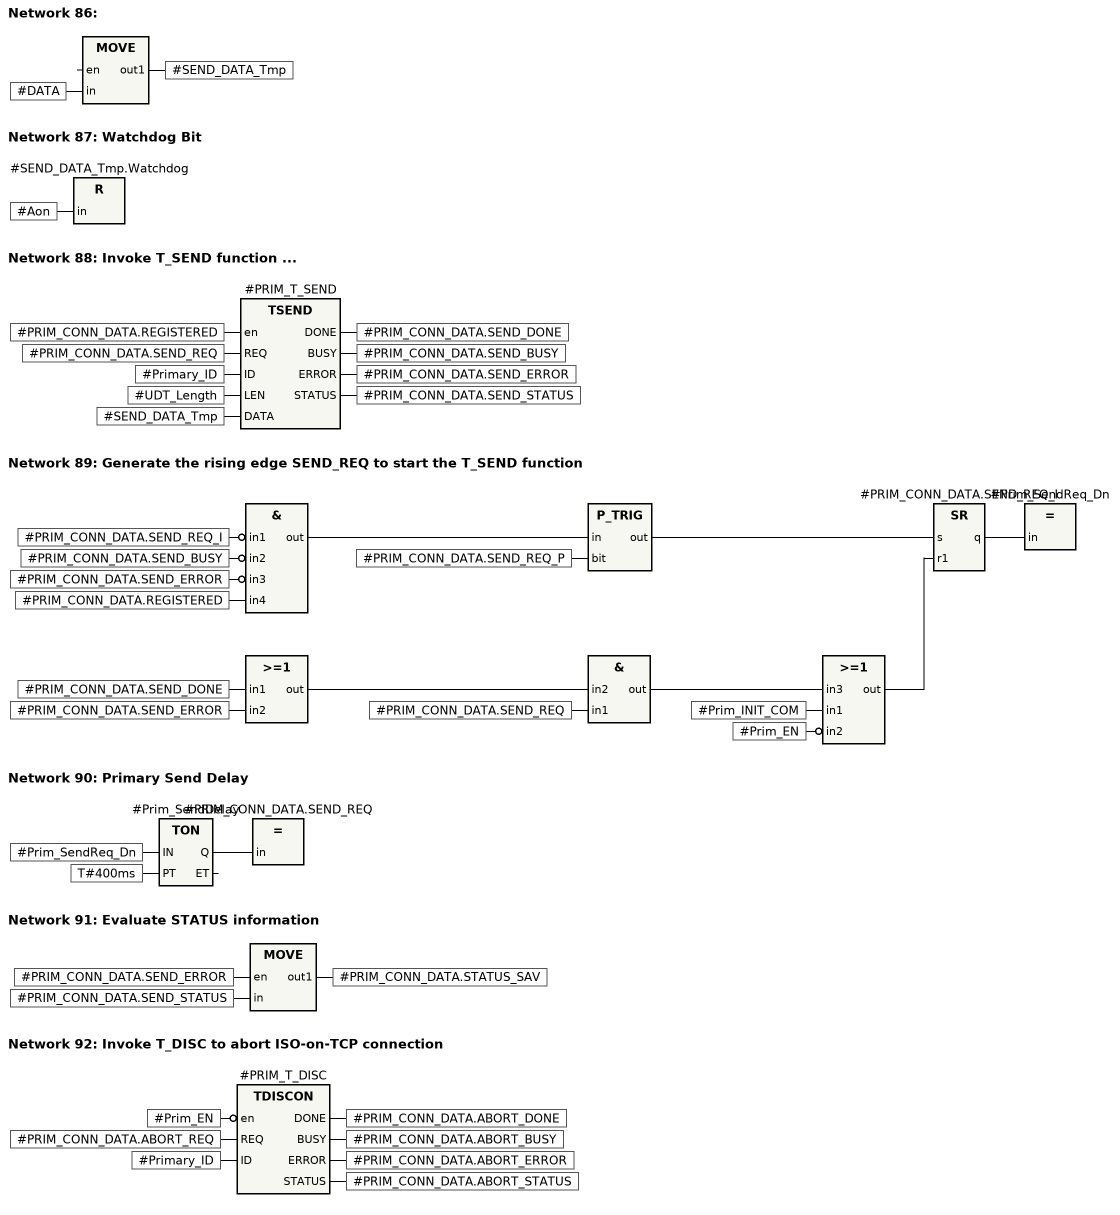
   #SEND_DATA_Tmp := #DATA;
END_REGION

REGION Network 87: Watchdog Bit
   IF #Aon THEN #SEND_DATA_Tmp.Watchdog := FALSE; END_IF;
END_REGION

REGION Network 88: Invoke T_SEND function ...
   // if connection is established to transmit the data to the partner as a message.
   IF #PRIM_CONN_DATA.REGISTERED THEN
       #PRIM_T_SEND(REQ := #PRIM_CONN_DATA.SEND_REQ,   // TSEND
                    ID := #Primary_ID,
                    LEN := #UDT_Length,
                    DATA := #SEND_DATA_Tmp,
                    DONE => #PRIM_CONN_DATA.SEND_DONE,
                    BUSY => #PRIM_CONN_DATA.SEND_BUSY,
                    ERROR => #PRIM_CONN_DATA.SEND_ERROR,
                    STATUS => #PRIM_CONN_DATA.SEND_STATUS);
   END_IF;
END_REGION

REGION Network 89: Generate the rising edge SEND_REQ to start the T_SEND function
   // Build002 - 27 March 2019 : Reset Condition Changed and Coil flag changed
   #_w1 := NOT #PRIM_CONN_DATA.SEND_REQ_I AND NOT #PRIM_CONN_DATA.SEND_BUSY AND NOT #PRIM_CONN_DATA.SEND_ERROR AND #PRIM_CONN_DATA.REGISTERED;
   #_w2 := #_w1 AND NOT #PRIM_CONN_DATA.SEND_REQ_P;   // rising edge
   #PRIM_CONN_DATA.SEND_REQ_P := #_w1;
   IF #_w2 THEN
       #PRIM_CONN_DATA.SEND_REQ_I := TRUE;   // SR flip-flop
   END_IF;
   IF ((#PRIM_CONN_DATA.SEND_DONE OR #PRIM_CONN_DATA.SEND_ERROR) AND #PRIM_CONN_DATA.SEND_REQ) OR #Prim_INIT_COM OR NOT #Prim_EN THEN
       #PRIM_CONN_DATA.SEND_REQ_I := FALSE;
   END_IF;
   #Prim_SendReq_Dn := #PRIM_CONN_DATA.SEND_REQ_I;
END_REGION

REGION Network 90: Primary Send Delay
   // Build002 - 27 March 2019 : Network Added
   #Prim_SendDelay(IN := #Prim_SendReq_Dn, PT := T#400ms);   // TON
   #PRIM_CONN_DATA.SEND_REQ := #Prim_SendDelay.Q;
END_REGION

REGION Network 91: Evaluate STATUS information
   // If ERROR occured then save STATUS!
   IF #PRIM_CONN_DATA.SEND_ERROR THEN #PRIM_CONN_DATA.STATUS_SAV := #PRIM_CONN_DATA.SEND_STATUS; END_IF;
END_REGION

REGION Network 92: Invoke T_DISC to abort ISO-on-TCP connection
   // The FB 66 "TDISCON" terminates a communications connection from the CPU to a
   // communications partner.
   // 
   // An existing connection is terminated when FB 66 "TDISCON" is called or when the
   // CPU has gone into STOP mode. To reestablish the connection, the FB 65 "TCON" 
   // has to be invoked again.
   IF NOT #Prim_EN THEN
       #PRIM_T_DISC(REQ := #PRIM_CONN_DATA.ABORT_REQ,   // TDISCON
                    ID := #Primary_ID,
                    DONE => #PRIM_CONN_DATA.ABORT_DONE,
                    BUSY => #PRIM_CONN_DATA.ABORT_BUSY,
                    ERROR => #PRIM_CONN_DATA.ABORT_ERROR,
                    STATUS => #PRIM_CONN_DATA.ABORT_STATUS);
   END_IF;
END_REGION

REGION Network 93: If "ABORT" is set, the connection will be aborted
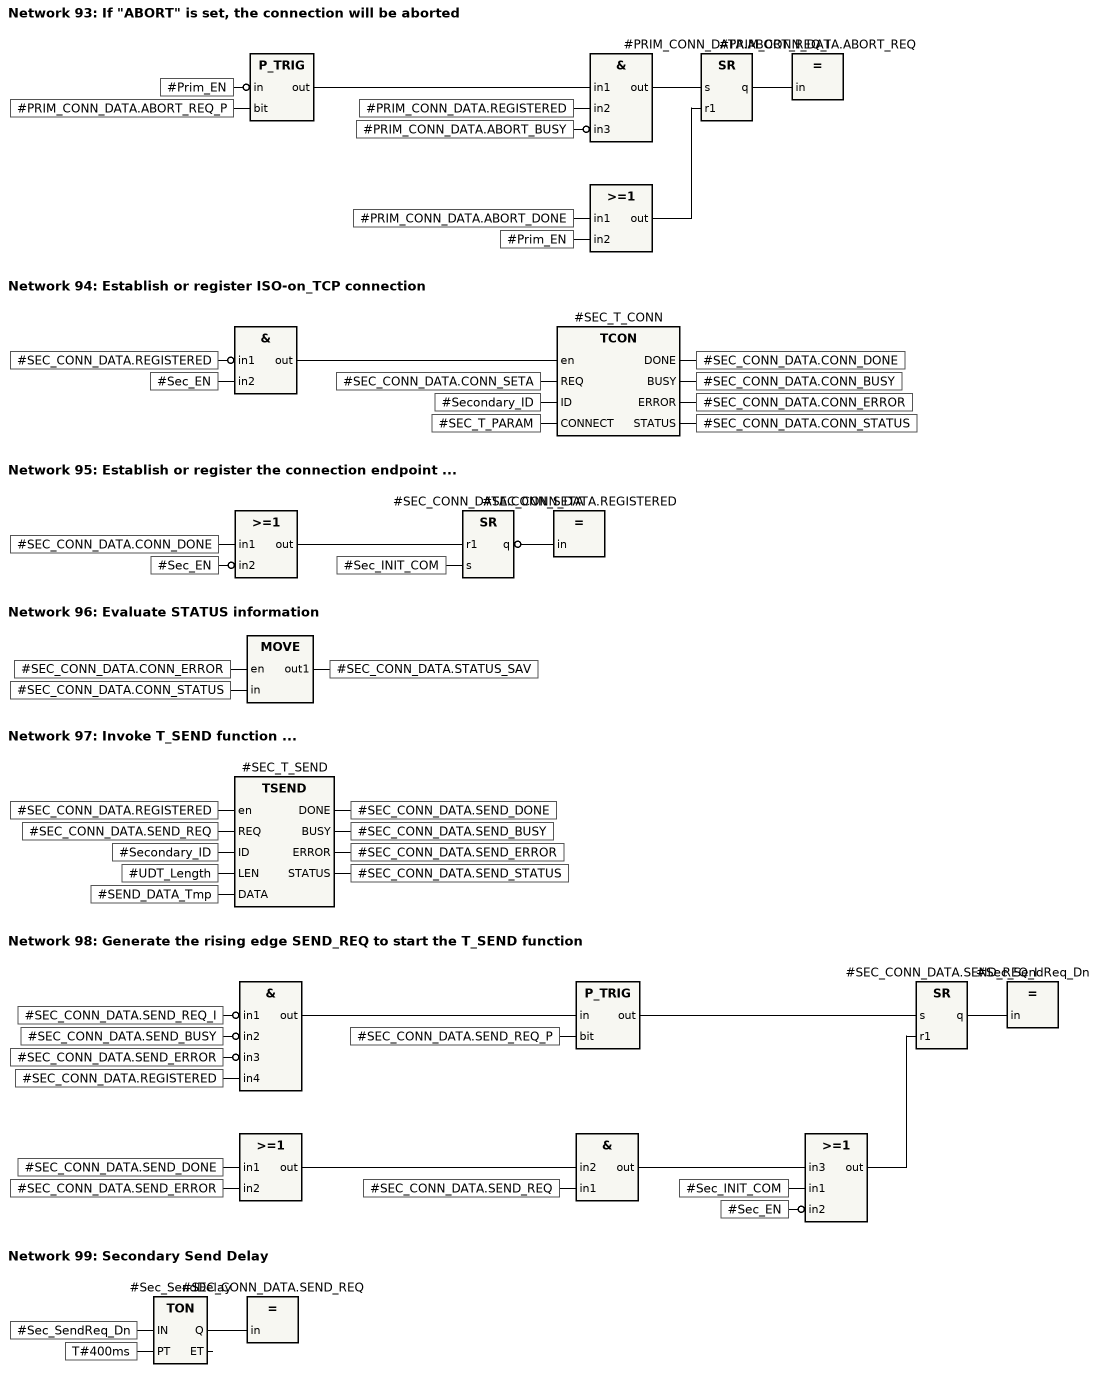
   #_w1 := NOT #Prim_EN AND NOT #PRIM_CONN_DATA.ABORT_REQ_P;   // rising edge
   #PRIM_CONN_DATA.ABORT_REQ_P := NOT #Prim_EN;
   IF #_w1 AND #PRIM_CONN_DATA.REGISTERED AND NOT #PRIM_CONN_DATA.ABORT_BUSY THEN
       #PRIM_CONN_DATA.ABORT_REQ_I := TRUE;   // SR flip-flop
   END_IF;
   IF #PRIM_CONN_DATA.ABORT_DONE OR #Prim_EN THEN #PRIM_CONN_DATA.ABORT_REQ_I := FALSE; END_IF;
   #PRIM_CONN_DATA.ABORT_REQ := #PRIM_CONN_DATA.ABORT_REQ_I;
END_REGION

REGION Network 94: Establish or register ISO-on_TCP connection
   // After the connection has been established, it is automatically monitored and 
   // maintained by the operating system of the CPU.
   // 
   // If the connection has been interrupted, by any line break or due to the remote 
   // communications partner, the active partner attempts to reestablish the 
   // connection.
   // 
   // Therefore, the FB 65 "TCON" may not be called again!
   IF NOT #SEC_CONN_DATA.REGISTERED AND #Sec_EN THEN
       #SEC_T_CONN(REQ := #SEC_CONN_DATA.CONN_SETA,   // TCON
                   ID := #Secondary_ID,
                   CONNECT := #SEC_T_PARAM,
                   DONE => #SEC_CONN_DATA.CONN_DONE,
                   BUSY => #SEC_CONN_DATA.CONN_BUSY,
                   ERROR => #SEC_CONN_DATA.CONN_ERROR,
                   STATUS => #SEC_CONN_DATA.CONN_STATUS);
   END_IF;
END_REGION

REGION Network 95: Establish or register the connection endpoint ...
   // while startup phase (initial).
   // 
   // Indication of the connection status:
   // 
   // a) If the CPU may establish the specified connection after Stop/Run  
   // immediately, the variable "REGISTERED" indicates HIGH (=1).
   // 
   // b) If the CPU is not able to establish the specified connection after Stop/Run, 
   // the variable "REGISTERED" remains LOW(=0).
   // 
   // c) Note: If the instance DB is loaded by the user, the variable "REGISTERED" 
   // indicates HIGH, although the connection may not be established yet. 
   // However, the FB64 "TRCV" would indicate the STATUS=0x80C4, as long as the 
   // connection has not been established.
   IF #Sec_INIT_COM THEN
       #SEC_CONN_DATA.CONN_SETA := TRUE;   // SR flip-flop
   END_IF;
   IF #SEC_CONN_DATA.CONN_DONE OR NOT #Sec_EN THEN #SEC_CONN_DATA.CONN_SETA := FALSE; END_IF;
   #SEC_CONN_DATA.REGISTERED := NOT #SEC_CONN_DATA.CONN_SETA;
END_REGION

REGION Network 96: Evaluate STATUS information
   // If ERROR occured then save STATUS!
   IF #SEC_CONN_DATA.CONN_ERROR THEN #SEC_CONN_DATA.STATUS_SAV := #SEC_CONN_DATA.CONN_STATUS; END_IF;
END_REGION

REGION Network 97: Invoke T_SEND function ...
   // if connection is established to transmit the data to the partner as a message.
   IF #SEC_CONN_DATA.REGISTERED THEN
       #SEC_T_SEND(REQ := #SEC_CONN_DATA.SEND_REQ,   // TSEND
                   ID := #Secondary_ID,
                   LEN := #UDT_Length,
                   DATA := #SEND_DATA_Tmp,
                   DONE => #SEC_CONN_DATA.SEND_DONE,
                   BUSY => #SEC_CONN_DATA.SEND_BUSY,
                   ERROR => #SEC_CONN_DATA.SEND_ERROR,
                   STATUS => #SEC_CONN_DATA.SEND_STATUS);
   END_IF;
END_REGION

REGION Network 98: Generate the rising edge SEND_REQ to start the T_SEND function
   // Build002 - 27 March 2019 : Reset Condition Changed and Coil flag changed
   #_w1 := NOT #SEC_CONN_DATA.SEND_REQ_I AND NOT #SEC_CONN_DATA.SEND_BUSY AND NOT #SEC_CONN_DATA.SEND_ERROR AND #SEC_CONN_DATA.REGISTERED;
   #_w2 := #_w1 AND NOT #SEC_CONN_DATA.SEND_REQ_P;   // rising edge
   #SEC_CONN_DATA.SEND_REQ_P := #_w1;
   IF #_w2 THEN
       #SEC_CONN_DATA.SEND_REQ_I := TRUE;   // SR flip-flop
   END_IF;
   IF ((#SEC_CONN_DATA.SEND_DONE OR #SEC_CONN_DATA.SEND_ERROR) AND #SEC_CONN_DATA.SEND_REQ) OR #Sec_INIT_COM OR NOT #Sec_EN THEN
       #SEC_CONN_DATA.SEND_REQ_I := FALSE;
   END_IF;
   #Sec_SendReq_Dn := #SEC_CONN_DATA.SEND_REQ_I;
END_REGION

REGION Network 99: Secondary Send Delay
   // Build002 - 27 March 2019 : Network Added
   #Sec_SendDelay(IN := #Sec_SendReq_Dn, PT := T#400ms);   // TON
   #SEC_CONN_DATA.SEND_REQ := #Sec_SendDelay.Q;
END_REGION

REGION Network 100: Evaluate STATUS information
   // If ERROR occured then save STATUS!
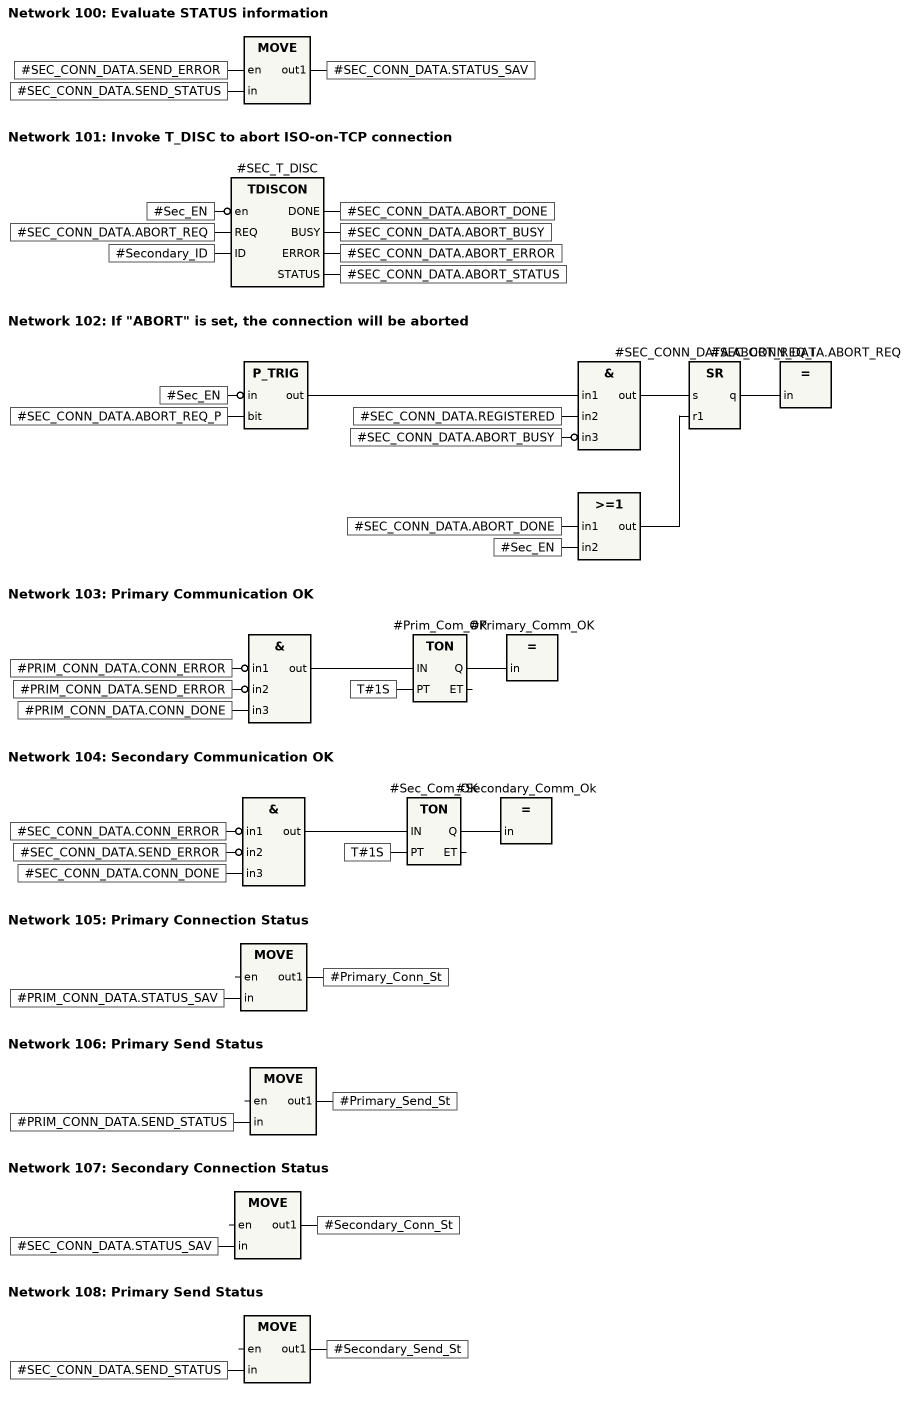
   IF #SEC_CONN_DATA.SEND_ERROR THEN #SEC_CONN_DATA.STATUS_SAV := #SEC_CONN_DATA.SEND_STATUS; END_IF;
END_REGION

REGION Network 101: Invoke T_DISC to abort ISO-on-TCP connection
   // The FB 66 "TDISCON" terminates a communications connection from the CPU to a
   // communications partner.
   // 
   // An existing connection is terminated when FB 66 "TDISCON" is called or when the
   // CPU has gone into STOP mode. To reestablish the connection, the FB 65 "TCON" 
   // has to be invoked again.
   IF NOT #Sec_EN THEN
       #SEC_T_DISC(REQ := #SEC_CONN_DATA.ABORT_REQ,   // TDISCON
                   ID := #Secondary_ID,
                   DONE => #SEC_CONN_DATA.ABORT_DONE,
                   BUSY => #SEC_CONN_DATA.ABORT_BUSY,
                   ERROR => #SEC_CONN_DATA.ABORT_ERROR,
                   STATUS => #SEC_CONN_DATA.ABORT_STATUS);
   END_IF;
END_REGION

REGION Network 102: If "ABORT" is set, the connection will be aborted
   #_w1 := NOT #Sec_EN AND NOT #SEC_CONN_DATA.ABORT_REQ_P;   // rising edge
   #SEC_CONN_DATA.ABORT_REQ_P := NOT #Sec_EN;
   IF #_w1 AND #SEC_CONN_DATA.REGISTERED AND NOT #SEC_CONN_DATA.ABORT_BUSY THEN
       #SEC_CONN_DATA.ABORT_REQ_I := TRUE;   // SR flip-flop
   END_IF;
   IF #SEC_CONN_DATA.ABORT_DONE OR #Sec_EN THEN #SEC_CONN_DATA.ABORT_REQ_I := FALSE; END_IF;
   #SEC_CONN_DATA.ABORT_REQ := #SEC_CONN_DATA.ABORT_REQ_I;
END_REGION

REGION Network 103: Primary Communication OK
   #Prim_Com_OK(IN := NOT #PRIM_CONN_DATA.CONN_ERROR AND NOT #PRIM_CONN_DATA.SEND_ERROR AND #PRIM_CONN_DATA.CONN_DONE,   // TON
                PT := T#1S);
   #Primary_Comm_OK := #Prim_Com_OK.Q;
END_REGION

REGION Network 104: Secondary Communication OK
   #Sec_Com_OK(IN := NOT #SEC_CONN_DATA.CONN_ERROR AND NOT #SEC_CONN_DATA.SEND_ERROR AND #SEC_CONN_DATA.CONN_DONE,   // TON
               PT := T#1S);
   #Secondary_Comm_Ok := #Sec_Com_OK.Q;
END_REGION

REGION Network 105: Primary Connection Status
   #Primary_Conn_St := #PRIM_CONN_DATA.STATUS_SAV;
END_REGION

REGION Network 106: Primary Send Status
   #Primary_Send_St := #PRIM_CONN_DATA.SEND_STATUS;
END_REGION

REGION Network 107: Secondary Connection Status
   #Secondary_Conn_St := #SEC_CONN_DATA.STATUS_SAV;
END_REGION

REGION Network 108: Primary Send Status
   #Secondary_Send_St := #SEC_CONN_DATA.SEND_STATUS;
END_REGION

REGION Network 109: Enable output ENO
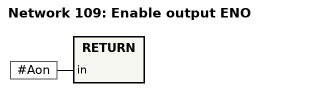
   IF #Aon THEN
       ENO := TRUE;
       RETURN;
   END_IF;
END_REGION
END_FUNCTION_BLOCK

FUNCTION_BLOCK "ACESYS_RCV"   // FB226, FBD
TITLE = ACESYS V8.0 - Build 002 - RECEIVE FUNCTION BLOCK
{ S7_Optimized_Access := 'TRUE' }
VERSION : 0.1
   VAR_INPUT
      Primary_EN : Bool;   // Enable Primary Link
      Primary_ID : Word;   // Valid from W#16#0001 to W#16#0FFF
      Primary_DEV_ID : Byte;   // 1 = Onboard (X1), 2 = Onboard (X2), 3 = Onboard (X3), 10 = External Cards
      Primary_ACT : Bool;   // ACTIVE=1; PASSIVE=0
      Primary_IP_ADDR1 : Int;
      Primary_IP_ADDR2 : Int;
      Primary_IP_ADDR3 : Int;
      Primary_IP_ADDR4 : Int;
      Primary_LOC_RS : Byte := BYTE#16#02;
      Primary_CP_RS : Byte;
      Primary_REM_RS : Byte := BYTE#16#02;
      Secondary_EN : Bool;   // Enable Secondary Link
      Secondary_ID : Word;   // Valid from W#16#0001 to W#16#0FFF
      Secondary_DEV_ID : Byte;   // B#16#01-IM151-8PN, #02-CPU31x-2PN/DP, #03-CPU319-3PN/DP, #05-CPU41x-3PN/DP
      Secondary_ACT : Bool;
      Secondary_IP_ADDR1 : Int;   // Secondary IP Address
      Secondary_IP_ADDR2 : Int;   // Secondary IP Address
      Secondary_IP_ADDR3 : Int;   // Secondary IP Address
      Secondary_IP_ADDR4 : Int;   // Secondary IP Address
      Secondary_LOC_RS : Byte := BYTE#16#02;   // Secondary Local Rack/Slot
      Secondary_CP_RS : Byte;   // Secondary CP Rack/Slot
      Secondary_REM_RS : Byte := BYTE#16#02;   // Secondary Remote Rack/Slot
      Clear_Bool : Bool;   // Clear Boolean Variables in case of Comm.Fault
      Clear_Int : Bool;   // Clear Integer Variables in case of Comm.Fault
      Clear_Real : Bool;   // Clear Real Variables in case of Comm.Fault
      MASTER_LINK : "ACESYS_MASTER_LINK";
   END_VAR
   VAR_OUTPUT
      Primary_Comm_OK : Bool;   // Primary Communication OK
      Primary_Conn_St : Word;   // Primary Connection Status
      Primary_Recv_St : Word;   // Primary Receive Status
      Secondary_Comm_Ok : Bool;   // Secondary Communication OK
      Secondary_Conn_St : Word;   // Secondary Connection Status
      Secondary_Recv_St : Word;   // Secondary Receive Status
      RCV_OK : Bool;   // Recive Data OK
      DATA : "ACESYS_PlcToPLC";
      MSW : "ACESYS_HMI_STAT_32T";
   END_VAR
   VAR
      BlockInfo : Struct
         Ace_Version : Int;   // Acesys Block Version Number
         Ace_BuildNo : Int;   // Acesys Block Build Number
         DB_Number : Int;   // Block Instance DB Number
      END_STRUCT;
      FP_CMD : Struct   // Faceplate Commands
         Spare_08 : Bool;
         Spare_09 : Bool;
         Spare_10 : Bool;
         Spare_11 : Bool;
         Spare_12 : Bool;
         Spare_13 : Bool;
         Spare_14 : Bool;
         AckAlarm : Bool;   // Alarm Acknowledge
         Spare_00 : Bool;
         Spare_01 : Bool;
         Spare_02 : Bool;
         Spare_03 : Bool;
         Spare_04 : Bool;
         Spare_05 : Bool;
         Spare_06 : Bool;
         Spare_07 : Bool;
      END_STRUCT;
      FP_PARM : Struct   // Faceplate Parameters
         Watchdog_PRE : Int := 5;   // Watchdog Time
         Watchdog_ACC : Int;   // Watchdog Time
      END_STRUCT;
      PRIM_RECV_DATA : "ACESYS_PlcToPLC";
      SEC_RECV_DATA : "ACESYS_PlcToPLC";
      PRIM_T_RECV : TRCV;
      PRIM_T_CONN : TCON;
      PRIM_T_DISC : TDISCON;
      PRIM_T_PARAM : TCON_IP_RFC;
      SEC_T_RECV : TRCV;
      SEC_T_CONN : TCON;
      SEC_T_DISC : TDISCON;
      SEC_T_PARAM : TCON_IP_RFC;
      PRIM_CONN_DATA : Struct
         REGISTERED : Bool;
         CONN_DONE : Bool;
         CONN_BUSY : Bool;
         CONN_ERROR : Bool;
         CONN_SETA : Bool;
         DISCONNECT : Bool;
         CONN_STATUS : Word;
         STATUS_SAV : Int;
         RECV_NDR : Bool;
         RECV_BUSY : Bool;
         RECV_ERROR : Bool;
         RECV_STATUS : Word;
         RECV_LEN : Int;
         RECV_LEN_S : Int;
         ABORT_REQ : Bool;
         ABORT_DONE : Bool;
         ABORT_BUSY : Bool;
         ABORT_ERROR : Bool;
         ABORT_REQ_I : Bool;
         ABORT_REQ_P : Bool;
         ABORT_STATUS : Word;
      END_STRUCT;
      SEC_CONN_DATA : Struct
         REGISTERED : Bool;
         CONN_DONE : Bool;
         CONN_BUSY : Bool;
         CONN_ERROR : Bool;
         CONN_SETA : Bool;
         DISCONNECT : Bool;
         CONN_STATUS : Word;
         STATUS_SAV : Int;
         RECV_NDR : Bool;
         RECV_BUSY : Bool;
         RECV_ERROR : Bool;
         RECV_STATUS : Word;
         RECV_LEN : Int;
         RECV_LEN_S : Int;
         ABORT_REQ : Bool;
         ABORT_DONE : Bool;
         ABORT_BUSY : Bool;
         ABORT_ERROR : Bool;
         ABORT_REQ_I : Bool;
         ABORT_REQ_P : Bool;
         ABORT_STATUS : Word;
      END_STRUCT;
      TSAP16 : String[16];
      ID AT TSAP16 : Array[1..18] of Byte;
      Prim_String : String[16];
      Sec_String : String[16];
      Watchdog_TimerMEM : Int;
      StatusWork : Int;
      AlarmNo : Int;
      AlarmNo_Old : Int;
      MSW_Status_Trans : Int;
      Primary_ID_Old : Word;
      Secondary_ID_Old : Word;
      CMD_Acknowledge : Bool;   // Internal Acknowledge
      Prim_INIT_COM : Bool;
      Sec_INIT_COM : Bool;
      Prim_En_ONS : Bool;
      Sec_En_ONS : Bool;
      Prim_Enabled_ONS : Bool;
      Sec_Enabled_ONS : Bool;
      SPECIFIED : Bool;
      Watchdog_TimerDN : Bool;
      Prim_ReCon_Active : Bool;   // Reconection Acive
      Sec_ReCon_Active : Bool;   // Reconection Acive
      ALARM_AlarmPresent : Bool;
      ALARM_WarnPresent : Bool;
      ALARM_Failure_Ack_Requ : Bool;
      ALARM_Warn_Ack_Required : Bool;
      Primary_Connect : Bool;   // Conect Primary Link
      Secondary_Connect : Bool;   // Conect Secondary Link
      Prim_Del_ReCon : TON_TIME;   // Delay Before Auto ReCone
      Prim_Con_TMR : TON_TIME;
      Sec_Del_ReCon : TON_TIME;   // Delay Before Auto ReConect
      Sec_Con_TMR : TON_TIME;
      Prim_Com_OK : TON_TIME;
      Sec_Com_OK : TON_TIME;
      PRIM_EXT_HWID : GEOADDR;
      SEC_EXT_HWID : GEOADDR;
      Out : Struct
         Primary_Comm_Ok : Bool;
         Secondary_Comm_Ok : Bool;
         RCV_OK : Bool;
         MSW_AlarmFailUnAck : Bool;
         Spare01 : Bool;
         Spare02 : Bool;
         Spare03 : Bool;
         Spare04 : Bool;
         Spare05 : Bool;
      END_STRUCT;
   END_VAR
   VAR_TEMP
      Aon : Bool;
      AOff : Bool;
      DummyBool : Bool;
      LOC_LEN : Int;
      REM_LEN : Int;
      TMP_INT : Int;
      LOC_RS : Int;
      TMP_RS : Int;
      TMP_DEV : Int;
      DummyDInt : DInt;
      RET : Int;
      UDT_Length : Int;
      t_Zero : Int;
      b_Zero : Array[0..1] of Byte;
   END_VAR
   VAR_TEMP   // added for the SCL form of the ladder/FBD networks
      _w1 : Bool;
      _w2 : Bool;
      _w3 : Bool;
   END_VAR
BEGIN

REGION Network 1: Aon
   // Acesys Receive Function Block based on Open Communication standard blocks FB64 
   // and FB65 for ISO-on-TCP
   // 
   // //////////////////////////////////////////////////////////////////////////////
   // 30/September/2014
   // Build 0: Block Start
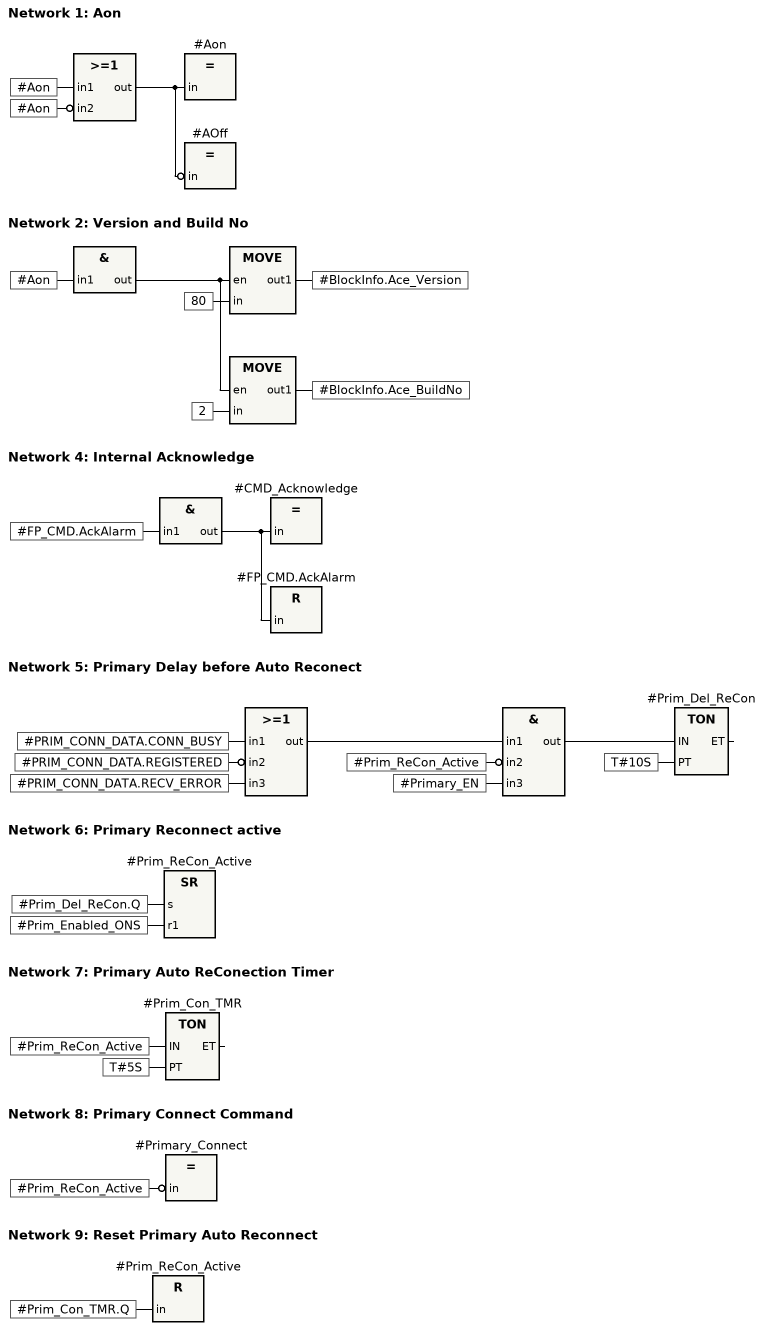
   #Aon := #Aon OR NOT #Aon;
   #AOff := NOT #Aon;
END_REGION

REGION Network 2: Version and Build No
   IF #Aon THEN
       #BlockInfo.Ace_Version := 80;
       #BlockInfo.Ace_BuildNo := 2;
   END_IF;
END_REGION

REGION Network 3 (STL): Instance DB Number to Faceplate
         L     DINO;
         T     #BlockInfo.DB_Number;
END_REGION

REGION Network 4: Internal Acknowledge
   // >>>>>>>Automatic Dep_CMD when use of block interface<<<<<<
   #CMD_Acknowledge := #FP_CMD.AckAlarm;
   IF #FP_CMD.AckAlarm THEN #FP_CMD.AckAlarm := FALSE; END_IF;
END_REGION

REGION Network 5: Primary Delay before Auto Reconect
   #Prim_Del_ReCon(IN := (#PRIM_CONN_DATA.CONN_BUSY OR NOT #PRIM_CONN_DATA.REGISTERED OR #PRIM_CONN_DATA.RECV_ERROR) AND NOT #Prim_ReCon_Active AND #Primary_EN,   // TON
                   PT := T#10S);
END_REGION

REGION Network 6: Primary Reconnect active
   IF #Prim_Del_ReCon.Q THEN
       #Prim_ReCon_Active := TRUE;   // SR flip-flop
   END_IF;
   IF #Prim_Enabled_ONS THEN #Prim_ReCon_Active := FALSE; END_IF;
END_REGION

REGION Network 7: Primary Auto ReConection Timer
   #Prim_Con_TMR(IN := #Prim_ReCon_Active, PT := T#5S);   // TON
END_REGION

REGION Network 8: Primary Connect Command
   #Primary_Connect := NOT #Prim_ReCon_Active;
END_REGION

REGION Network 9: Reset Primary Auto Reconnect
   IF #Prim_Con_TMR.Q THEN #Prim_ReCon_Active := FALSE; END_IF;
END_REGION

REGION Network 10: Skip if Primay Enable is True
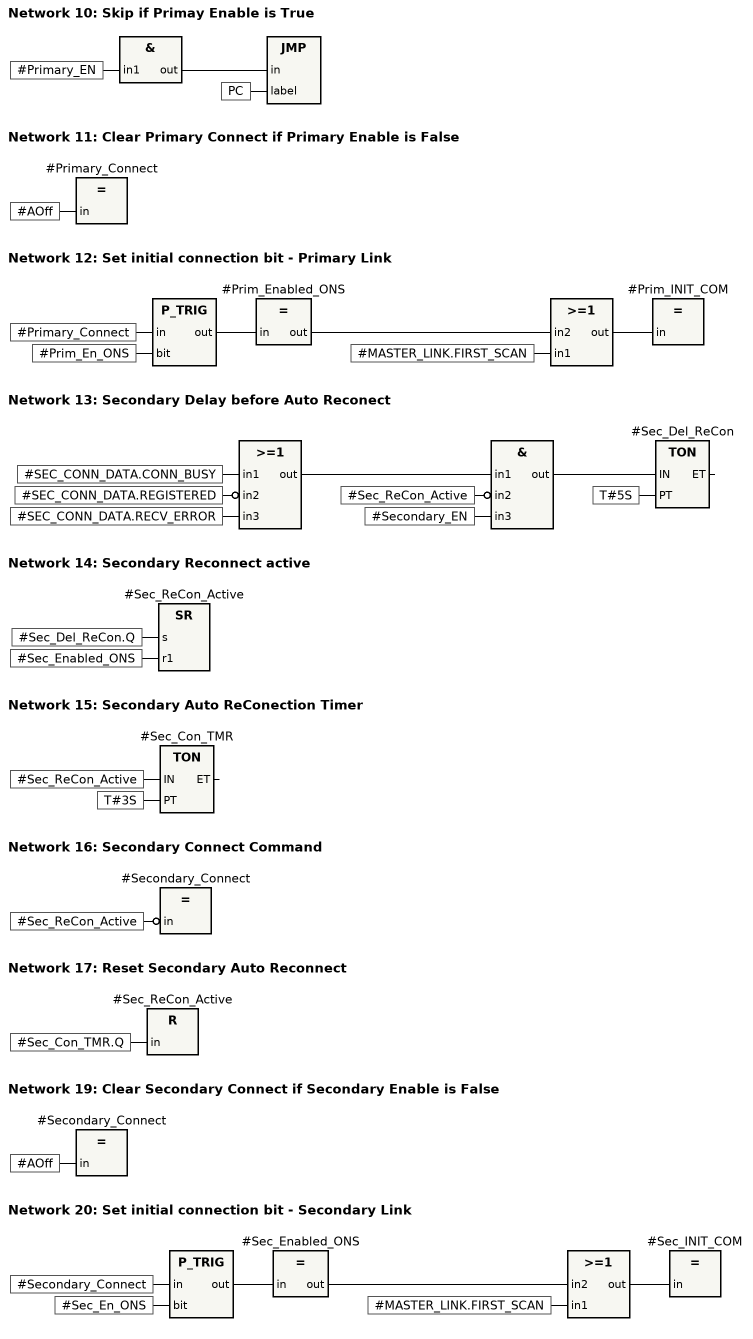
   IF #Primary_EN THEN GOTO PC; END_IF;
END_REGION

REGION Network 11: Clear Primary Connect if Primary Enable is False
   #Primary_Connect := #AOff;
END_REGION

REGION Network 12: Set initial connection bit - Primary Link
   PC:
   #_w1 := #Primary_Connect AND NOT #Prim_En_ONS;   // rising edge
   #Prim_En_ONS := #Primary_Connect;
   #Prim_Enabled_ONS := #_w1;
   #Prim_INIT_COM := #_w1 OR #MASTER_LINK.FIRST_SCAN;
END_REGION

REGION Network 13: Secondary Delay before Auto Reconect
   #Sec_Del_ReCon(IN := (#SEC_CONN_DATA.CONN_BUSY OR NOT #SEC_CONN_DATA.REGISTERED OR #SEC_CONN_DATA.RECV_ERROR) AND NOT #Sec_ReCon_Active AND #Secondary_EN,   // TON
                  PT := T#5S);
END_REGION

REGION Network 14: Secondary Reconnect active
   IF #Sec_Del_ReCon.Q THEN
       #Sec_ReCon_Active := TRUE;   // SR flip-flop
   END_IF;
   IF #Sec_Enabled_ONS THEN #Sec_ReCon_Active := FALSE; END_IF;
END_REGION

REGION Network 15: Secondary Auto ReConection Timer
   #Sec_Con_TMR(IN := #Sec_ReCon_Active, PT := T#3S);   // TON
END_REGION

REGION Network 16: Secondary Connect Command
   #Secondary_Connect := NOT #Sec_ReCon_Active;
END_REGION

REGION Network 17: Reset Secondary Auto Reconnect
   IF #Sec_Con_TMR.Q THEN #Sec_ReCon_Active := FALSE; END_IF;
END_REGION

REGION Network 18 (STL): Skip if Secondary Enable is True
         A     #Secondary_EN;
         JC    SC;
END_REGION

REGION Network 19: Clear Secondary Connect if Secondary Enable is False
   #Secondary_Connect := #AOff;
END_REGION

REGION Network 20: Set initial connection bit - Secondary Link
   SC:
   #_w1 := #Secondary_Connect AND NOT #Sec_En_ONS;   // rising edge
   #Sec_En_ONS := #Secondary_Connect;
   #Sec_Enabled_ONS := #_w1;
   #Sec_INIT_COM := #_w1 OR #MASTER_LINK.FIRST_SCAN;
END_REGION

REGION Network 21: Clear Bits to start initial connection and communication
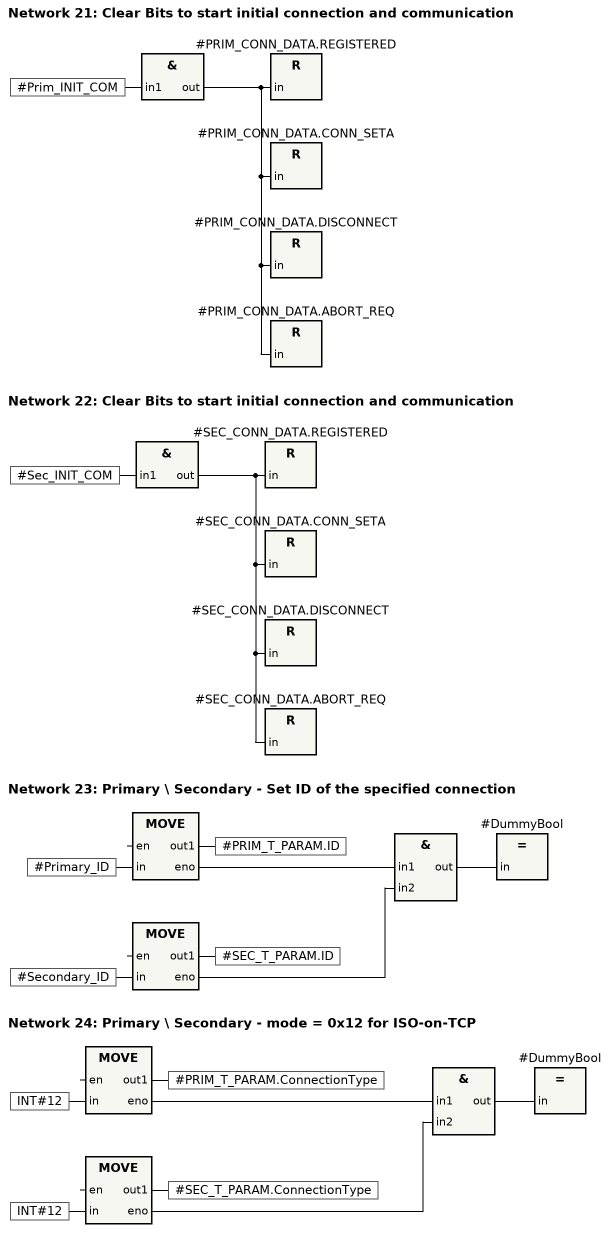
   IF #Prim_INIT_COM THEN
       #PRIM_CONN_DATA.REGISTERED := FALSE;
       #PRIM_CONN_DATA.CONN_SETA := FALSE;
       #PRIM_CONN_DATA.DISCONNECT := FALSE;
       #PRIM_CONN_DATA.ABORT_REQ := FALSE;
   END_IF;
END_REGION

REGION Network 22: Clear Bits to start initial connection and communication
   IF #Sec_INIT_COM THEN
       #SEC_CONN_DATA.REGISTERED := FALSE;
       #SEC_CONN_DATA.CONN_SETA := FALSE;
       #SEC_CONN_DATA.DISCONNECT := FALSE;
       #SEC_CONN_DATA.ABORT_REQ := FALSE;
   END_IF;
END_REGION

REGION Network 23: Primary \ Secondary - Set ID of the specified connection
   // ENO of a box is taken as its EN; it also drops when the box reports an error
   #PRIM_T_PARAM.ID := #Primary_ID;
   #SEC_T_PARAM.ID := #Secondary_ID;
   #DummyBool := TRUE;
END_REGION

REGION Network 24: Primary \ Secondary - mode = 0x12 for ISO-on-TCP
   // ENO of a box is taken as its EN; it also drops when the box reports an error
   #PRIM_T_PARAM.ConnectionType := INT#12;
   #SEC_T_PARAM.ConnectionType := INT#12;
   #DummyBool := TRUE;
END_REGION

REGION Network 25: <<<<<<<< PRIMARY >>>>>>>>
END_REGION

REGION Network 26: Hardware Identifier OnBoard
   // Build 002 viv-in 15 Feb 2022 -  X2 Port number corrected.
